LIN {X 0,Y 159.433,Z 807.885,A -85,B 0,C 180,E1 -24356.561,E2 -24356.561} C_VEL
LIN {X 0,Y 155.614,Z 816.206,A -85,B 0,C 180,E1 -24359.65,E2 -24359.65} C_VEL
LIN {X 0,Y 151.771,Z 823.644,A -85,B 0,C 180,E1 -24363.159,E2 -24363.159} C_VEL
LIN {X 0,Y 148.83,Z 828.918,A -85,B 0,C 180,E1 -24366.333,E2 -24366.333} C_VEL
LIN {X 0,Y 145.963,Z 834.064,A -85,B 0,C 180,E1 -24370.301,E2 -24370.301} C_VEL
LIN {X 0,Y 143.724,Z 838.04,A -85,B 0,C 180,E1 -24374.396,E2 -24374.396} C_VEL
LIN {X 0,Y 142.137,Z 840.967,A -85,B 0,C 180,E1 -24378.591,E2 -24378.591} C_VEL
LIN {X 0,Y 141.434,Z 842.382,A -85,B 0,C 180,E1 -24381.425,E2 -24381.425} C_VEL
LIN {X 0,Y 140.7,Z 843.984,A -85,B 0,C 180,E1 -24387.135,E2 -24387.135} C_VEL
LIN {X 0,Y 140.69,Z 844.211,A -85,B 0,C 180,E1 -24389.998,E2 -24389.998} C_VEL
LIN {X 0,Y 140.947,Z 843.425,A -85,B 0,C 180,E1 -24395.721,E2 -24395.721} C_VEL
LIN {X 0,Y 141.432,Z 842.454,A -85,B 0,C 180,E1 -24398.571,E2 -24398.571} C_VEL
LIN {X 0,Y 142.132,Z 841.08,A -85,B 0,C 180,E1 -24401.405,E2 -24401.405} C_VEL
LIN {X 0,Y 143.688,Z 838.194,A -85,B 0,C 180,E1 -24405.603,E2 -24405.603} C_VEL
LIN {X 0,Y 145.898,Z 834.266,A -85,B 0,C 180,E1 -24409.703,E2 -24409.703} C_VEL
LIN {X 0,Y 148.753,Z 829.176,A -85,B 0,C 180,E1 -24413.675,E2 -24413.675} C_VEL
LIN {X 0,Y 152.357,Z 822.754,A -85,B 0,C 180,E1 -24417.467,E2 -24417.467} C_VEL
LIN {X 0,Y 156.625,Z 814.287,A -85,B 0,C 180,E1 -24421.308,E2 -24421.308} C_VEL
LIN {X 0,Y 160.109,Z 806.58,A -85,B 0,C 180,E1 -24424.029,E2 -24424.029} C_VEL
LIN {X 0,Y 164.319,Z 796.492,A -85,B 0,C 180,E1 -24426.78,E2 -24426.78} C_VEL
LIN {X 0,Y 168.42,Z 785.143,A -85,B 0,C 180,E1 -24429.132,E2 -24429.132} C_VEL
LIN {X 0,Y 171.709,Z 773.906,A -85,B 0,C 180,E1 -24430.907,E2 -24430.907} C_VEL
LIN {X 0,Y 174.569,Z 761.518,A -85,B 0,C 180,E1 -24432.338,E2 -24432.338} C_VEL
LIN {X 0,Y 176.775,Z 748.935,A -85,B 0,C 180,E1 -24433.335,E2 -24433.335} C_VEL
LIN {X 0,Y 177.807,Z 738.757,A -85,B 0,C 180,E1 -24433.901,E2 -24433.901} C_VEL
LIN {X 0,Y 173.307,Z 740.765,A -85,B 0,C 180,E1 -24435.203,E2 -24435.203} C_VEL
LIN {X 0,Y 170.147,Z 741.611,A -85,B 0,C 180,E1 -24436.222,E2 -24436.222} C_VEL
LIN {X 0,Y 165.898,Z 744.296,A -85,B 0,C 180,E1 -24437.532,E2 -24437.532} C_VEL
LIN {X 0,Y 162.52,Z 745.361,A -85,B 0,C 180,E1 -24438.74,E2 -24438.74} C_VEL
LIN {X 0,Y 159.499,Z 745.547,A -85,B 0,C 180,E1 -24439.98,E2 -24439.98} C_VEL
LIN {X 0,Y 155.97,Z 747.642,A -85,B 0,C 180,E1 -24441.302,E2 -24441.302} C_VEL
LIN {X 0,Y 154.26,Z 748.147,A -85,B 0,C 180,E1 -24442.044,E2 -24442.044} C_VEL
LIN {X 0,Y 150.109,Z 747.859,A -85,B 0,C 180,E1 -24444.18,E2 -24444.18} C_VEL
LIN {X 0,Y 147.27,Z 749.37,A -85,B 0,C 180,E1 -24445.53,E2 -24445.53} C_VEL
LIN {X 0,Y 145.442,Z 749.393,A -85,B 0,C 180,E1 -24446.599,E2 -24446.599} C_VEL
LIN {X 0,Y 144.475,Z 748.528,A -85,B 0,C 180,E1 -24447.325,E2 -24447.325} C_VEL
LIN {X 0,Y 144.158,Z 747.052,A -85,B 0,C 180,E1 -24447.828,E2 -24447.828} C_VEL
LIN {X 0,Y 143.492,Z 754.332,A -85,B 0,C 180,E1 -24451.83,E2 -24451.83} C_VEL
LIN {X 0,Y 143.482,Z 761.799,A -85,B 0,C 180,E1 -24456.93,E2 -24456.93} C_VEL
LIN {X 0,Y 144.233,Z 767.1,A -85,B 0,C 180,E1 -24461.535,E2 -24461.535} C_VEL
LIN {X 0,Y 145.804,Z 771.093,A -85,B 0,C 180,E1 -24466.054,E2 -24466.054} C_VEL
LIN {X 0,Y 147.276,Z 773.104,A -85,B 0,C 180,E1 -24468.996,E2 -24468.996} C_VEL
LIN {X 0,Y 149.078,Z 774.683,A -85,B 0,C 180,E1 -24471.869,E2 -24471.869} C_VEL
LIN {X 0,Y 151.257,Z 775.775,A -85,B 0,C 180,E1 -24474.668,E2 -24474.668} C_VEL
LIN {X 0,Y 154.674,Z 776.543,A -85,B 0,C 180,E1 -24478.326,E2 -24478.326} C_VEL
LIN {X 0,Y 159.556,Z 776.355,A -85,B 0,C 180,E1 -24482.524,E2 -24482.524} C_VEL
LIN {X 0,Y 162.872,Z 775.642,A -85,B 0,C 180,E1 -24484.951,E2 -24484.951} C_VEL
LIN {X 0,Y 166.498,Z 774.491,A -85,B 0,C 180,E1 -24487.275,E2 -24487.275} C_VEL
LIN {X 0,Y 171.25,Z 772.464,A -85,B 0,C 180,E1 -24489.971,E2 -24489.971} C_VEL
LIN {X 0,Y 176.597,Z 769.564,A -85,B 0,C 180,E1 -24492.643,E2 -24492.643} C_VEL
LIN {X 0,Y 183.317,Z 765.026,A -85,B 0,C 180,E1 -24495.567,E2 -24495.567} C_VEL
LIN {X 0,Y 190.412,Z 759.281,A -85,B 0,C 180,E1 -24498.284,E2 -24498.284} C_VEL
LIN {X 0,Y 197.891,Z 752.001,A -85,B 0,C 180,E1 -24500.802,E2 -24500.802} C_VEL
LIN {X 0,Y 205.676,Z 742.876,A -85,B 0,C 180,E1 -24503.14,E2 -24503.14} C_VEL
LIN {X 0,Y 212.006,Z 734.049,A -85,B 0,C 180,E1 -24504.884,E2 -24504.884} C_VEL
LIN {X 0,Y 217.692,Z 724.562,A -85,B 0,C 180,E1 -24506.354,E2 -24506.354} C_VEL
LIN {X 0,Y 223.591,Z 712.612,A -85,B 0,C 180,E1 -24507.824,E2 -24507.824} C_VEL
LIN {X 0,Y 228.396,Z 700.131,A -85,B 0,C 180,E1 -24508.987,E2 -24508.987} C_VEL
LIN {X 0,Y 231.612,Z 688.931,A -85,B 0,C 180,E1 -24509.841,E2 -24509.841} C_VEL
LIN {X 0,Y 232.53,Z 684.952,A -85,B 0,C 180,E1 -24510.119,E2 -24510.119} C_VEL
LIN {X 0,Y 232.21,Z 685.318,A -85,B 0,C 180,E1 -24511.425,E2 -24511.425} C_VEL
LIN {X 0,Y 231.811,Z 686.774,A -85,B 0,C 180,E1 -24512.878,E2 -24512.878} C_VEL
LIN {X 0,Y 231.448,Z 690.251,A -85,B 0,C 180,E1 -24515.018,E2 -24515.018} C_VEL
LIN {X 0,Y 228.723,Z 701.141,A -85,B 0,C 180,E1 -24515.936,E2 -24515.936} C_VEL
LIN {X 0,Y 223.27,Z 716.625,A -85,B 0,C 180,E1 -24516.732,E2 -24516.732} C_VEL
LIN {X 0,Y 217.31,Z 729.757,A -85,B 0,C 180,E1 -24517.598,E2 -24517.598} C_VEL
LIN {X 0,Y 211.644,Z 740.071,A -85,B 0,C 180,E1 -24518.504,E2 -24518.504} C_VEL
LIN {X 0,Y 208.404,Z 744.999,A -85,B 0,C 180,E1 -24518.827,E2 -24518.827} C_VEL
LIN {X 0,Y 202.208,Z 752.79,A -85,B 0,C 180,E1 -24518.994,E2 -24518.994} C_VEL
LIN {X 0,Y 195.68,Z 759.99,A -85,B 0,C 180,E1 -24519.3,E2 -24519.3} C_VEL
LIN {X 0,Y 191.955,Z 764.049,A -85,B 0,C 180,E1 -24519.853,E2 -24519.853} C_VEL
LIN {X 0,Y 182.386,Z 774.075,A -85,B 0,C 180,E1 -24522.121,E2 -24522.121} C_VEL
LIN {X 0,Y 173.174,Z 782.415,A -85,B 0,C 180,E1 -24524.751,E2 -24524.751} C_VEL
LIN {X 0,Y 165.897,Z 788.257,A -85,B 0,C 180,E1 -24527.33,E2 -24527.33} C_VEL
LIN {X 0,Y 162.05,Z 791.386,A -85,B 0,C 180,E1 -24529.011,E2 -24529.011} C_VEL
LIN {X 0,Y 157.677,Z 802.954,A -85,B 0,C 180,E1 -24531.394,E2 -24531.394} C_VEL
LIN {X 0,Y 153.161,Z 813.235,A -85,B 0,C 180,E1 -24534.197,E2 -24534.197} C_VEL
LIN {X 0,Y 149.036,Z 821.56,A -85,B 0,C 180,E1 -24537.163,E2 -24537.163} C_VEL
LIN {X 0,Y 144.79,Z 829.691,A -85,B 0,C 180,E1 -24540.965,E2 -24540.965} C_VEL
LIN {X 0,Y 141.114,Z 836.225,A -85,B 0,C 180,E1 -24544.958,E2 -24544.958} C_VEL
LIN {X 0,Y 138.146,Z 841.42,A -85,B 0,C 180,E1 -24549.141,E2 -24549.141} C_VEL
LIN {X 0,Y 135.89,Z 845.439,A -85,B 0,C 180,E1 -24553.477,E2 -24553.477} C_VEL
LIN {X 0,Y 134.464,Z 848.406,A -85,B 0,C 180,E1 -24557.935,E2 -24557.935} C_VEL
LIN {X 0,Y 133.856,Z 849.828,A -85,B 0,C 180,E1 -24560.94,E2 -24560.94} C_VEL
LIN {X 0,Y 133.526,Z 851.454,A -85,B 0,C 180,E1 -24566.985,E2 -24566.985} C_VEL
LIN {X 0,Y 133.661,Z 851.673,A -85,B 0,C 180,E1 -24570.003,E2 -24570.003} C_VEL
LIN {X 0,Y 133.527,Z 851.438,A -85,B 0,C 180,E1 -24573.02,E2 -24573.02} C_VEL
LIN {X 0,Y 133.558,Z 850.809,A -85,B 0,C 180,E1 -24576.044,E2 -24576.044} C_VEL
LIN {X 0,Y 133.858,Z 849.789,A -85,B 0,C 180,E1 -24579.065,E2 -24579.065} C_VEL
LIN {X 0,Y 134.464,Z 848.345,A -85,B 0,C 180,E1 -24582.07,E2 -24582.07} C_VEL
LIN {X 0,Y 135.87,Z 845.356,A -85,B 0,C 180,E1 -24586.531,E2 -24586.531} C_VEL
LIN {X 0,Y 138.113,Z 841.312,A -85,B 0,C 180,E1 -24590.869,E2 -24590.869} C_VEL
LIN {X 0,Y 141.693,Z 835.082,A -85,B 0,C 180,E1 -24595.724,E2 -24595.724} C_VEL
LIN {X 0,Y 145.364,Z 828.414,A -85,B 0,C 180,E1 -24599.629,E2 -24599.629} C_VEL
LIN {X 0,Y 148.981,Z 821.355,A -85,B 0,C 180,E1 -24602.856,E2 -24602.856} C_VEL
LIN {X 0,Y 153.1,Z 812.99,A -85,B 0,C 180,E1 -24605.825,E2 -24605.825} C_VEL
LIN {X 0,Y 157.64,Z 802.637,A -85,B 0,C 180,E1 -24608.622,E2 -24608.622} C_VEL
LIN {X 0,Y 162.078,Z 790.989,A -85,B 0,C 180,E1 -24610.986,E2 -24610.986} C_VEL
LIN {X 0,Y 165.633,Z 779.257,A -85,B 0,C 180,E1 -24612.76,E2 -24612.76} C_VEL
LIN {X 0,Y 168.637,Z 767.119,A -85,B 0,C 180,E1 -24614.065,E2 -24614.065} C_VEL
LIN {X 0,Y 170.976,Z 754.448,A -85,B 0,C 180,E1 -24614.98,E2 -24614.98} C_VEL
LIN {X 0,Y 172.29,Z 740.764,A -85,B 0,C 180,E1 -24615.626,E2 -24615.626} C_VEL
LIN {X 0,Y 175.16,Z 696.8,A -85,B 0,C 180,E1 -24617.207,E2 -24617.207} C_VEL
LIN {X 0,Y 174.375,Z 675.084,A -85,B 0,C 180,E1 -24618.793,E2 -24618.793} C_VEL
LIN {X 0,Y 172.801,Z 650.948,A -85,B 0,C 180,E1 -24620.919,E2 -24620.919} C_VEL
LIN {X 0,Y 171.783,Z 647.337,A -85,B 0,C 180,E1 -24621.573,E2 -24621.573} C_VEL
LIN {X 0,Y 168.493,Z 637.862,A -85,B 0,C 180,E1 -24623.661,E2 -24623.661} C_VEL
LIN {X 0,Y 164.617,Z 631.829,A -85,B 0,C 180,E1 -24626.032,E2 -24626.032} C_VEL
LIN {X 0,Y 161.633,Z 625.28,A -85,B 0,C 180,E1 -24629.999,E2 -24629.999} C_VEL
LIN {X 0,Y 160.602,Z 623.765,A -85,B 0,C 180,E1 -24631.225,E2 -24631.225} C_VEL
LIN {X 0,Y 158.998,Z 620.197,A -85,B 0,C 180,E1 -24633.767,E2 -24633.767} C_VEL
LIN {X 0,Y 156.671,Z 616.136,A -85,B 0,C 180,E1 -24637.586,E2 -24637.586} C_VEL
LIN {X 0,Y 154.772,Z 612.752,A -85,B 0,C 180,E1 -24641.466,E2 -24641.466} C_VEL
LIN {X 0,Y 152.828,Z 609.327,A -85,B 0,C 180,E1 -24646.707,E2 -24646.707} C_VEL
LIN {X 0,Y 151.398,Z 607.318,A -85,B 0,C 180,E1 -24651.995,E2 -24651.995} C_VEL
LIN {X 0,Y 150.986,Z 606.091,A -85,B 0,C 180,E1 -24657.332,E2 -24657.332} C_VEL
LIN {X 0,Y 151.07,Z 605.988,A -85,B 0,C 180,E1 -24660,E2 -24660} C_VEL
LIN {X 0,Y 151.49,Z 607.972,A -85,B 0,C 180,E1 -24668,E2 -24668} C_VEL
LIN {X 0,Y 151.967,Z 609.157,A -85,B 0,C 180,E1 -24670.661,E2 -24670.661} C_VEL
LIN {X 0,Y 153.211,Z 612.572,A -85,B 0,C 180,E1 -24675.976,E2 -24675.976} C_VEL
LIN {X 0,Y 154.985,Z 617.053,A -85,B 0,C 180,E1 -24681.271,E2 -24681.271} C_VEL
LIN {X 0,Y 156.601,Z 621.203,A -85,B 0,C 180,E1 -24685.236,E2 -24685.236} C_VEL
LIN {X 0,Y 158.276,Z 626.514,A -85,B 0,C 180,E1 -24689.238,E2 -24689.238} C_VEL
LIN {X 0,Y 159.234,Z 629.154,A -85,B 0,C 180,E1 -24690.99,E2 -24690.99} C_VEL
LIN {X 0,Y 163.41,Z 636.139,A -85,B 0,C 180,E1 -24693.902,E2 -24693.902} C_VEL
LIN {X 0,Y 167.489,Z 643.377,A -85,B 0,C 180,E1 -24696.449,E2 -24696.449} C_VEL
LIN {X 0,Y 173.046,Z 655.01,A -85,B 0,C 180,E1 -24699.63,E2 -24699.63} C_VEL
LIN {X 0,Y 175.92,Z 662.099,A -85,B 0,C 180,E1 -24701.184,E2 -24701.184} C_VEL
LIN {X 0,Y 177.008,Z 677.278,A -85,B 0,C 180,E1 -24702.491,E2 -24702.491} C_VEL
LIN {X 0,Y 172.398,Z 741.841,A -85,B 0,C 180,E1 -24704.776,E2 -24704.776} C_VEL
LIN {X 0,Y 170.625,Z 754.436,A -85,B 0,C 180,E1 -24705.553,E2 -24705.553} C_VEL
LIN {X 0,Y 168.07,Z 767.088,A -85,B 0,C 180,E1 -24706.783,E2 -24706.783} C_VEL
LIN {X 0,Y 165.024,Z 778.4,A -85,B 0,C 180,E1 -24708.282,E2 -24708.282} C_VEL
LIN {X 0,Y 161.571,Z 788.778,A -85,B 0,C 180,E1 -24710.087,E2 -24710.087} C_VEL
LIN {X 0,Y 157.386,Z 799.406,A -85,B 0,C 180,E1 -24712.523,E2 -24712.523} C_VEL
LIN {X 0,Y 152.732,Z 809.817,A -85,B 0,C 180,E1 -24715.687,E2 -24715.687} C_VEL
LIN {X 0,Y 148.959,Z 817.482,A -85,B 0,C 180,E1 -24718.734,E2 -24718.734} C_VEL
LIN {X 0,Y 144.814,Z 824.954,A -85,B 0,C 180,E1 -24722.543,E2 -24722.543} C_VEL
LIN {X 0,Y 141.194,Z 830.953,A -85,B 0,C 180,E1 -24726.532,E2 -24726.532} C_VEL
LIN {X 0,Y 138.391,Z 835.687,A -85,B 0,C 180,E1 -24730.723,E2 -24730.723} C_VEL
LIN {X 0,Y 136.233,Z 839.302,A -85,B 0,C 180,E1 -24735.05,E2 -24735.05} C_VEL
LIN {X 0,Y 135.172,Z 841.161,A -85,B 0,C 180,E1 -24737.994,E2 -24737.994} C_VEL
LIN {X 0,Y 134.428,Z 842.575,A -85,B 0,C 180,E1 -24740.974,E2 -24740.974} C_VEL
LIN {X 0,Y 133.633,Z 844.176,A -85,B 0,C 180,E1 -24746.983,E2 -24746.983} C_VEL
LIN {X 0,Y 133.57,Z 844.347,A -85,B 0,C 180,E1 -24751.354,E2 -24751.354} C_VEL
LIN {X 0,Y 133.882,Z 843.618,A -85,B 0,C 180,E1 -24756.024,E2 -24756.024} C_VEL
LIN {X 0,Y 134.426,Z 842.646,A -85,B 0,C 180,E1 -24759.021,E2 -24759.021} C_VEL
LIN {X 0,Y 135.167,Z 841.272,A -85,B 0,C 180,E1 -24762.001,E2 -24762.001} C_VEL
LIN {X 0,Y 136.845,Z 838.386,A -85,B 0,C 180,E1 -24766.405,E2 -24766.405} C_VEL
LIN {X 0,Y 139.231,Z 834.456,A -85,B 0,C 180,E1 -24770.689,E2 -24770.689} C_VEL
LIN {X 0,Y 142.276,Z 829.365,A -85,B 0,C 180,E1 -24774.824,E2 -24774.824} C_VEL
LIN {X 0,Y 146.084,Z 822.942,A -85,B 0,C 180,E1 -24778.754,E2 -24778.754} C_VEL
LIN {X 0,Y 150.335,Z 814.98,A -85,B 0,C 180,E1 -24782.501,E2 -24782.501} C_VEL
LIN {X 0,Y 154.286,Z 806.764,A -85,B 0,C 180,E1 -24785.502,E2 -24785.502} C_VEL
LIN {X 0,Y 158.687,Z 796.672,A -85,B 0,C 180,E1 -24788.315,E2 -24788.315} C_VEL
LIN {X 0,Y 162.977,Z 785.318,A -85,B 0,C 180,E1 -24790.706,E2 -24790.706} C_VEL
LIN {X 0,Y 166.409,Z 774.073,A -85,B 0,C 180,E1 -24792.507,E2 -24792.507} C_VEL
LIN {X 0,Y 169.354,Z 761.865,A -85,B 0,C 180,E1 -24793.935,E2 -24793.935} C_VEL
LIN {X 0,Y 171.675,Z 749.194,A -85,B 0,C 180,E1 -24794.947,E2 -24794.947} C_VEL
LIN {X 0,Y 171.743,Z 747.989,A -85,B 0,C 180,E1 -24795.061,E2 -24795.061} C_VEL
LIN {X 0,Y 170.353,Z 748.631,A -85,B 0,C 180,E1 -24795.465,E2 -24795.465} C_VEL
LIN {X 0,Y 165.327,Z 751.285,A -85,B 0,C 180,E1 -24796.936,E2 -24796.936} C_VEL
LIN {X 0,Y 161.312,Z 752.281,A -85,B 0,C 180,E1 -24798.363,E2 -24798.363} C_VEL
LIN {X 0,Y 159.242,Z 752.563,A -85,B 0,C 180,E1 -24799.176,E2 -24799.176} C_VEL
LIN {X 0,Y 154.898,Z 754.619,A -85,B 0,C 180,E1 -24800.774,E2 -24800.774} C_VEL
LIN {X 0,Y 152.892,Z 755.029,A -85,B 0,C 180,E1 -24801.643,E2 -24801.643} C_VEL
LIN {X 0,Y 149.193,Z 754.991,A -85,B 0,C 180,E1 -24803.507,E2 -24803.507} C_VEL
LIN {X 0,Y 146.355,Z 756.162,A -85,B 0,C 180,E1 -24804.813,E2 -24804.813} C_VEL
LIN {X 0,Y 144.323,Z 756.378,A -85,B 0,C 180,E1 -24805.943,E2 -24805.943} C_VEL
LIN {X 0,Y 141.694,Z 755.49,A -85,B 0,C 180,E1 -24807.778,E2 -24807.778} C_VEL
LIN {X 0,Y 139.146,Z 756.562,A -85,B 0,C 180,E1 -24809.243,E2 -24809.243} C_VEL
LIN {X 0,Y 137.107,Z 756.278,A -85,B 0,C 180,E1 -24810.803,E2 -24810.803} C_VEL
LIN {X 0,Y 136.443,Z 754.919,A -85,B 0,C 180,E1 -24811.661,E2 -24811.661} C_VEL
LIN {X 0,Y 136.386,Z 754.349,A -85,B 0,C 180,E1 -24811.846,E2 -24811.846} C_VEL
LIN {X 0,Y 136.282,Z 759.966,A -85,B 0,C 180,E1 -24815.634,E2 -24815.634} C_VEL
LIN {X 0,Y 136.88,Z 765.906,A -85,B 0,C 180,E1 -24820.504,E2 -24820.504} C_VEL
LIN {X 0,Y 138.319,Z 770.505,A -85,B 0,C 180,E1 -24825.282,E2 -24825.282} C_VEL
LIN {X 0,Y 139.725,Z 772.89,A -85,B 0,C 180,E1 -24828.393,E2 -24828.393} C_VEL
LIN {X 0,Y 141.912,Z 775.165,A -85,B 0,C 180,E1 -24832.06,E2 -24832.06} C_VEL
LIN {X 0,Y 146.128,Z 777.229,A -85,B 0,C 180,E1 -24837.243,E2 -24837.243} C_VEL
LIN {X 0,Y 148.914,Z 777.777,A -85,B 0,C 180,E1 -24840,E2 -24840} C_VEL
LIN {X 0,Y 152.048,Z 777.864,A -85,B 0,C 180,E1 -24842.649,E2 -24842.649} C_VEL
LIN {X 0,Y 155.449,Z 777.501,A -85,B 0,C 180,E1 -24845.188,E2 -24845.188} C_VEL
LIN {X 0,Y 159.131,Z 776.727,A -85,B 0,C 180,E1 -24847.614,E2 -24847.614} C_VEL
LIN {X 0,Y 164.484,Z 774.951,A -85,B 0,C 180,E1 -24850.678,E2 -24850.678} C_VEL
LIN {X 0,Y 171.757,Z 771.563,A -85,B 0,C 180,E1 -24854.212,E2 -24854.212} C_VEL
LIN {X 0,Y 178.839,Z 767.322,A -85,B 0,C 180,E1 -24857.142,E2 -24857.142} C_VEL
LIN {X 0,Y 187.16,Z 761.027,A -85,B 0,C 180,E1 -24860.162,E2 -24860.162} C_VEL
LIN {X 0,Y 195.403,Z 753.555,A -85,B 0,C 180,E1 -24862.746,E2 -24862.746} C_VEL
LIN {X 0,Y 203.187,Z 744.927,A -85,B 0,C 180,E1 -24864.922,E2 -24864.922} C_VEL
LIN {X 0,Y 211.228,Z 734.197,A -85,B 0,C 180,E1 -24866.958,E2 -24866.958} C_VEL
LIN {X 0,Y 217.505,Z 723.948,A -85,B 0,C 180,E1 -24868.451,E2 -24868.451} C_VEL
LIN {X 0,Y 222.732,Z 713.501,A -85,B 0,C 180,E1 -24869.651,E2 -24869.651} C_VEL
LIN {X 0,Y 227.729,Z 700.942,A -85,B 0,C 180,E1 -24870.781,E2 -24870.781} C_VEL
LIN {X 0,Y 230.426,Z 692.352,A -85,B 0,C 180,E1 -24871.455,E2 -24871.455} C_VEL
LIN {X 0,Y 230.064,Z 693.596,A -85,B 0,C 180,E1 -24872.512,E2 -24872.512} C_VEL
LIN {X 0,Y 229.618,Z 695.562,A -85,B 0,C 180,E1 -24873.654,E2 -24873.654} C_VEL
LIN {X 0,Y 227,Z 704.287,A -85,B 0,C 180,E1 -24874.323,E2 -24874.323} C_VEL
LIN {X 0,Y 221.503,Z 718.33,A -85,B 0,C 180,E1 -24875.011,E2 -24875.011} C_VEL
LIN {X 0,Y 214.736,Z 731.889,A -85,B 0,C 180,E1 -24875.905,E2 -24875.905} C_VEL
LIN {X 0,Y 206.968,Z 744.59,A -85,B 0,C 180,E1 -24877.066,E2 -24877.066} C_VEL
LIN {X 0,Y 199.435,Z 755.069,A -85,B 0,C 180,E1 -24878.368,E2 -24878.368} C_VEL
LIN {X 0,Y 191.955,Z 764.049,A -85,B 0,C 180,E1 -24879.853,E2 -24879.853} C_VEL
LIN {X 0,Y 188.055,Z 768.042,A -85,B 0,C 180,E1 -24880.484,E2 -24880.484} C_VEL
LIN {X 0,Y 180.591,Z 774.245,A -85,B 0,C 180,E1 -24881.156,E2 -24881.156} C_VEL
LIN {X 0,Y 172.911,Z 779.836,A -85,B 0,C 180,E1 -24881.995,E2 -24881.995} C_VEL
LIN {X 0,Y 168.724,Z 782.875,A -85,B 0,C 180,E1 -24882.91,E2 -24882.91} C_VEL
LIN {X 0,Y 160.759,Z 788.694,A -85,B 0,C 180,E1 -24885.619,E2 -24885.619} C_VEL
LIN {X 0,Y 156.614,Z 791.561,A -85,B 0,C 180,E1 -24887.369,E2 -24887.369} C_VEL
LIN {X 0,Y 152.177,Z 802.773,A -85,B 0,C 180,E1 -24889.721,E2 -24889.721} C_VEL
LIN {X 0,Y 147.436,Z 813.051,A -85,B 0,C 180,E1 -24892.575,E2 -24892.575} C_VEL
LIN {X 0,Y 142.306,Z 822.849,A -85,B 0,C 180,E1 -24896.252,E2 -24896.252} C_VEL
LIN {X 0,Y 137.863,Z 830.844,A -85,B 0,C 180,E1 -24900.289,E2 -24900.289} C_VEL
LIN {X 0,Y 134.701,Z 836.035,A -85,B 0,C 180,E1 -24903.677,E2 -24903.677} C_VEL
LIN {X 0,Y 131.506,Z 841.228,A -85,B 0,C 180,E1 -24908.035,E2 -24908.035} C_VEL
LIN {X 0,Y 129.067,Z 845.246,A -85,B 0,C 180,E1 -24912.576,E2 -24912.576} C_VEL
LIN {X 0,Y 127.491,Z 848.213,A -85,B 0,C 180,E1 -24917.264,E2 -24917.264} C_VEL
LIN {X 0,Y 126.82,Z 849.635,A -85,B 0,C 180,E1 -24920.433,E2 -24920.433} C_VEL
LIN {X 0,Y 126.445,Z 851.261,A -85,B 0,C 180,E1 -24926.816,E2 -24926.816} C_VEL
LIN {X 0,Y 126.514,Z 851.446,A -85,B 0,C 180,E1 -24930.718,E2 -24930.718} C_VEL
LIN {X 0,Y 126.476,Z 850.615,A -85,B 0,C 180,E1 -24936.383,E2 -24936.383} C_VEL
LIN {X 0,Y 126.822,Z 849.595,A -85,B 0,C 180,E1 -24939.572,E2 -24939.572} C_VEL
LIN {X 0,Y 127.489,Z 848.15,A -85,B 0,C 180,E1 -24942.741,E2 -24942.741} C_VEL
LIN {X 0,Y 129.045,Z 845.162,A -85,B 0,C 180,E1 -24947.432,E2 -24947.432} C_VEL
LIN {X 0,Y 131.479,Z 841.118,A -85,B 0,C 180,E1 -24951.976,E2 -24951.976} C_VEL
LIN {X 0,Y 135.331,Z 834.889,A -85,B 0,C 180,E1 -24957.029,E2 -24957.029} C_VEL
LIN {X 0,Y 139.29,Z 828.099,A -85,B 0,C 180,E1 -24961.145,E2 -24961.145} C_VEL
LIN {X 0,Y 143.051,Z 821.164,A -85,B 0,C 180,E1 -24964.403,E2 -24964.403} C_VEL
LIN {X 0,Y 147.384,Z 812.8,A -85,B 0,C 180,E1 -24967.446,E2 -24967.446} C_VEL
LIN {X 0,Y 152.149,Z 802.45,A -85,B 0,C 180,E1 -24970.294,E2 -24970.294} C_VEL
LIN {X 0,Y 156.785,Z 790.806,A -85,B 0,C 180,E1 -24972.689,E2 -24972.689} C_VEL
LIN {X 0,Y 160.501,Z 779.079,A -85,B 0,C 180,E1 -24974.478,E2 -24974.478} C_VEL
LIN {X 0,Y 163.621,Z 766.951,A -85,B 0,C 180,E1 -24975.791,E2 -24975.791} C_VEL
LIN {X 0,Y 166.018,Z 754.47,A -85,B 0,C 180,E1 -24976.698,E2 -24976.698} C_VEL
LIN {X 0,Y 167.449,Z 740.25,A -85,B 0,C 180,E1 -24977.371,E2 -24977.371} C_VEL
LIN {X 0,Y 170.376,Z 697.159,A -85,B 0,C 180,E1 -24978.946,E2 -24978.946} C_VEL
LIN {X 0,Y 169.601,Z 673.672,A -85,B 0,C 180,E1 -24980.756,E2 -24980.756} C_VEL
LIN {X 0,Y 168.379,Z 653.086,A -85,B 0,C 180,E1 -24982.657,E2 -24982.657} C_VEL
LIN {X 0,Y 164.983,Z 642.689,A -85,B 0,C 180,E1 -24984.988,E2 -24984.988} C_VEL
LIN {X 0,Y 160.526,Z 635.959,A -85,B 0,C 180,E1 -24987.868,E2 -24987.868} C_VEL
LIN {X 0,Y 157.768,Z 631.739,A -85,B 0,C 180,E1 -24989.924,E2 -24989.924} C_VEL
LIN {X 0,Y 154.856,Z 625.663,A -85,B 0,C 180,E1 -24994.46,E2 -24994.46} C_VEL
LIN {X 0,Y 152.595,Z 621.59,A -85,B 0,C 180,E1 -24998.38,E2 -24998.38} C_VEL
LIN {X 0,Y 151.362,Z 619.266,A -85,B 0,C 180,E1 -25001.033,E2 -25001.033} C_VEL
LIN {X 0,Y 149.279,Z 615.652,A -85,B 0,C 180,E1 -25006.385,E2 -25006.385} C_VEL
LIN {X 0,Y 147.929,Z 613.563,A -85,B 0,C 180,E1 -25011.806,E2 -25011.806} C_VEL
LIN {X 0,Y 147.441,Z 612.273,A -85,B 0,C 180,E1 -25017.268,E2 -25017.268} C_VEL
LIN {X 0,Y 147.42,Z 612.095,A -85,B 0,C 180,E1 -25020,E2 -25020} C_VEL
LIN {X 0,Y 147.709,Z 614.109,A -85,B 0,C 180,E1 -25028.207,E2 -25028.207} C_VEL
LIN {X 0,Y 148.616,Z 616.961,A -85,B 0,C 180,E1 -25033.677,E2 -25033.677} C_VEL
LIN {X 0,Y 150.103,Z 621.034,A -85,B 0,C 180,E1 -25039.132,E2 -25039.132} C_VEL
LIN {X 0,Y 151.554,Z 624.94,A -85,B 0,C 180,E1 -25043.215,E2 -25043.215} C_VEL
LIN {X 0,Y 153.161,Z 629.484,A -85,B 0,C 180,E1 -25046.987,E2 -25046.987} C_VEL
LIN {X 0,Y 157.861,Z 637.183,A -85,B 0,C 180,E1 -25050.855,E2 -25050.855} C_VEL
LIN {X 0,Y 162.168,Z 644.72,A -85,B 0,C 180,E1 -25053.916,E2 -25053.916} C_VEL
LIN {X 0,Y 166.718,Z 654,A -85,B 0,C 180,E1 -25056.845,E2 -25056.845} C_VEL
LIN {X 0,Y 170.665,Z 663.158,A -85,B 0,C 180,E1 -25059.188,E2 -25059.188} C_VEL
LIN {X 0,Y 171.442,Z 665.479,A -85,B 0,C 180,E1 -25059.656,E2 -25059.656} C_VEL
LIN {X 0,Y 172.284,Z 677.342,A -85,B 0,C 180,E1 -25060.745,E2 -25060.745} C_VEL
LIN {X 0,Y 167.532,Z 741.504,A -85,B 0,C 180,E1 -25063.035,E2 -25063.035} C_VEL
LIN {X 0,Y 165.64,Z 754.6,A -85,B 0,C 180,E1 -25063.836,E2 -25063.836} C_VEL
LIN {X 0,Y 162.977,Z 767.264,A -85,B 0,C 180,E1 -25065.077,E2 -25065.077} C_VEL
LIN {X 0,Y 159.801,Z 778.581,A -85,B 0,C 180,E1 -25066.59,E2 -25066.59} C_VEL
LIN {X 0,Y 156.205,Z 788.963,A -85,B 0,C 180,E1 -25068.42,E2 -25068.42} C_VEL
LIN {X 0,Y 151.816,Z 799.594,A -85,B 0,C 180,E1 -25070.893,E2 -25070.893} C_VEL
LIN {X 0,Y 146.926,Z 810.008,A -85,B 0,C 180,E1 -25074.127,E2 -25074.127} C_VEL
LIN {X 0,Y 142.152,Z 819.012,A -85,B 0,C 180,E1 -25077.892,E2 -25077.892} C_VEL
LIN {X 0,Y 137.908,Z 826.24,A -85,B 0,C 180,E1 -25081.873,E2 -25081.873} C_VEL
LIN {X 0,Y 134.702,Z 831.146,A -85,B 0,C 180,E1 -25085.327,E2 -25085.327} C_VEL
LIN {X 0,Y 131.702,Z 835.88,A -85,B 0,C 180,E1 -25089.702,E2 -25089.702} C_VEL
LIN {X 0,Y 129.377,Z 839.495,A -85,B 0,C 180,E1 -25094.237,E2 -25094.237} C_VEL
LIN {X 0,Y 128.235,Z 841.355,A -85,B 0,C 180,E1 -25097.334,E2 -25097.334} C_VEL
LIN {X 0,Y 127.415,Z 842.768,A -85,B 0,C 180,E1 -25100.473,E2 -25100.473} C_VEL
LIN {X 0,Y 126.555,Z 844.369,A -85,B 0,C 180,E1 -25106.814,E2 -25106.814} C_VEL
LIN {X 0,Y 126.505,Z 844.597,A -85,B 0,C 180,E1 -25109.997,E2 -25109.997} C_VEL
LIN {X 0,Y 126.515,Z 844.4,A -85,B 0,C 180,E1 -25113.182,E2 -25113.182} C_VEL
LIN {X 0,Y 127.412,Z 842.839,A -85,B 0,C 180,E1 -25119.522,E2 -25119.522} C_VEL
LIN {X 0,Y 128.23,Z 841.465,A -85,B 0,C 180,E1 -25122.661,E2 -25122.661} C_VEL
LIN {X 0,Y 130.034,Z 838.578,A -85,B 0,C 180,E1 -25127.29,E2 -25127.29} C_VEL
LIN {X 0,Y 132.589,Z 834.648,A -85,B 0,C 180,E1 -25131.777,E2 -25131.777} C_VEL
LIN {X 0,Y 135.863,Z 829.555,A -85,B 0,C 180,E1 -25136.081,E2 -25136.081} C_VEL
LIN {X 0,Y 139.892,Z 823.131,A -85,B 0,C 180,E1 -25140.155,E2 -25140.155} C_VEL
LIN {X 0,Y 144.129,Z 815.654,A -85,B 0,C 180,E1 -25143.805,E2 -25143.805} C_VEL
LIN {X 0,Y 148.549,Z 806.948,A -85,B 0,C 180,E1 -25147.097,E2 -25147.097} C_VEL
LIN {X 0,Y 153.171,Z 796.852,A -85,B 0,C 180,E1 -25149.965,E2 -25149.965} C_VEL
LIN {X 0,Y 157.677,Z 785.493,A -85,B 0,C 180,E1 -25152.385,E2 -25152.385} C_VEL
LIN {X 0,Y 161.248,Z 774.239,A -85,B 0,C 180,E1 -25154.212,E2 -25154.212} C_VEL
LIN {X 0,Y 164.213,Z 762.493,A -85,B 0,C 180,E1 -25155.605,E2 -25155.605} C_VEL
LIN {X 0,Y 164.872,Z 759.472,A -85,B 0,C 180,E1 -25155.902,E2 -25155.902} C_VEL
LIN {X 0,Y 164.837,Z 758.01,A -85,B 0,C 180,E1 -25156.145,E2 -25156.145} C_VEL
LIN {X 0,Y 158.589,Z 759.444,A -85,B 0,C 180,E1 -25158.337,E2 -25158.337} C_VEL
LIN {X 0,Y 153.51,Z 761.453,A -85,B 0,C 180,E1 -25160.137,E2 -25160.137} C_VEL
LIN {X 0,Y 149.078,Z 761.696,A -85,B 0,C 180,E1 -25162.203,E2 -25162.203} C_VEL
LIN {X 0,Y 144.566,Z 762.932,A -85,B 0,C 180,E1 -25164.311,E2 -25164.311} C_VEL
LIN {X 0,Y 140.685,Z 762.736,A -85,B 0,C 180,E1 -25166.666,E2 -25166.666} C_VEL
LIN {X 0,Y 136.805,Z 763.364,A -85,B 0,C 180,E1 -25169.088,E2 -25169.088} C_VEL
LIN {X 0,Y 133.746,Z 762.181,A -85,B 0,C 180,E1 -25171.775,E2 -25171.775} C_VEL
LIN {X 0,Y 130.379,Z 762.932,A -85,B 0,C 180,E1 -25174.454,E2 -25174.454} C_VEL
LIN {X 0,Y 129.322,Z 761.702,A -85,B 0,C 180,E1 -25175.948,E2 -25175.948} C_VEL
LIN {X 0,Y 129.256,Z 760.809,A -85,B 0,C 180,E1 -25176.461,E2 -25176.461} C_VEL
LIN {X 0,Y 129.865,Z 766.248,A -85,B 0,C 180,E1 -25181.052,E2 -25181.052} C_VEL
LIN {X 0,Y 131.559,Z 771.297,A -85,B 0,C 180,E1 -25186.348,E2 -25186.348} C_VEL
LIN {X 0,Y 133.882,Z 774.659,A -85,B 0,C 180,E1 -25190.939,E2 -25190.939} C_VEL
LIN {X 0,Y 136.005,Z 776.458,A -85,B 0,C 180,E1 -25194.068,E2 -25194.068} C_VEL
LIN {X 0,Y 140.563,Z 778.488,A -85,B 0,C 180,E1 -25199.281,E2 -25199.281} C_VEL
LIN {X 0,Y 144.502,Z 779.122,A -85,B 0,C 180,E1 -25202.788,E2 -25202.788} C_VEL
LIN {X 0,Y 148.31,Z 779.089,A -85,B 0,C 180,E1 -25205.689,E2 -25205.689} C_VEL
LIN {X 0,Y 151.734,Z 778.683,A -85,B 0,C 180,E1 -25207.987,E2 -25207.987} C_VEL
LIN {X 0,Y 157.752,Z 777.23,A -85,B 0,C 180,E1 -25211.459,E2 -25211.459} C_VEL
LIN {X 0,Y 164.645,Z 774.685,A -85,B 0,C 180,E1 -25214.84,E2 -25214.84} C_VEL
LIN {X 0,Y 171.963,Z 771.028,A -85,B 0,C 180,E1 -25217.85,E2 -25217.85} C_VEL
LIN {X 0,Y 180.574,Z 765.56,A -85,B 0,C 180,E1 -25220.926,E2 -25220.926} C_VEL
LIN {X 0,Y 188.994,Z 758.942,A -85,B 0,C 180,E1 -25223.563,E2 -25223.563} C_VEL
LIN {X 0,Y 197.431,Z 750.915,A -85,B 0,C 180,E1 -25225.853,E2 -25225.853} C_VEL
LIN {X 0,Y 205.459,Z 741.705,A -85,B 0,C 180,E1 -25227.807,E2 -25227.807} C_VEL
LIN {X 0,Y 212.612,Z 731.752,A -85,B 0,C 180,E1 -25229.446,E2 -25229.446} C_VEL
LIN {X 0,Y 219.241,Z 720.541,A -85,B 0,C 180,E1 -25230.857,E2 -25230.857} C_VEL
LIN {X 0,Y 224.436,Z 709.655,A -85,B 0,C 180,E1 -25231.925,E2 -25231.925} C_VEL
LIN {X 0,Y 225.949,Z 705.881,A -85,B 0,C 180,E1 -25232.24,E2 -25232.24} C_VEL
LIN {X 0,Y 225.364,Z 707.49,A -85,B 0,C 180,E1 -25232.653,E2 -25232.653} C_VEL
LIN {X 0,Y 219.384,Z 721.166,A -85,B 0,C 180,E1 -25233.325,E2 -25233.325} C_VEL
LIN {X 0,Y 212.339,Z 734.087,A -85,B 0,C 180,E1 -25234.166,E2 -25234.166} C_VEL
LIN {X 0,Y 204.416,Z 746.084,A -85,B 0,C 180,E1 -25235.264,E2 -25235.264} C_VEL
LIN {X 0,Y 195.145,Z 757.762,A -85,B 0,C 180,E1 -25236.748,E2 -25236.748} C_VEL
LIN {X 0,Y 186.286,Z 767.447,A -85,B 0,C 180,E1 -25238.483,E2 -25238.483} C_VEL
LIN {X 0,Y 176.339,Z 776.656,A -85,B 0,C 180,E1 -25240.782,E2 -25240.782} C_VEL
LIN {X 0,Y 168.724,Z 782.875,A -85,B 0,C 180,E1 -25242.91,E2 -25242.91} C_VEL
LIN {X 0,Y 164.599,Z 785.76,A -85,B 0,C 180,E1 -25243.921,E2 -25243.921} C_VEL
LIN {X 0,Y 157.089,Z 790.755,A -85,B 0,C 180,E1 -25245.244,E2 -25245.244} C_VEL
LIN {X 0,Y 151.584,Z 795.369,A -85,B 0,C 180,E1 -25246.268,E2 -25246.268} C_VEL
LIN {X 0,Y 148.373,Z 799.439,A -85,B 0,C 180,E1 -25247.182,E2 -25247.182} C_VEL
LIN {X 0,Y 147.592,Z 800.923,A -85,B 0,C 180,E1 -25247.531,E2 -25247.531} C_VEL
LIN {X 0,Y 142.816,Z 810.957,A -85,B 0,C 180,E1 -25250.232,E2 -25250.232} C_VEL
LIN {X 0,Y 138.153,Z 819.646,A -85,B 0,C 180,E1 -25253.296,E2 -25253.296} C_VEL
LIN {X 0,Y 134.025,Z 826.814,A -85,B 0,C 180,E1 -25256.595,E2 -25256.595} C_VEL
LIN {X 0,Y 129.75,Z 833.841,A -85,B 0,C 180,E1 -25260.828,E2 -25260.828} C_VEL
LIN {X 0,Y 125.999,Z 839.43,A -85,B 0,C 180,E1 -25265.274,E2 -25265.274} C_VEL
LIN {X 0,Y 123.022,Z 843.815,A -85,B 0,C 180,E1 -25269.958,E2 -25269.958} C_VEL
LIN {X 0,Y 121.624,Z 846.132,A -85,B 0,C 180,E1 -25273.21,E2 -25273.21} C_VEL
LIN {X 0,Y 120.547,Z 848.02,A -85,B 0,C 180,E1 -25276.517,E2 -25276.517} C_VEL
LIN {X 0,Y 119.808,Z 849.442,A -85,B 0,C 180,E1 -25279.867,E2 -25279.867} C_VEL
LIN {X 0,Y 119.356,Z 851.068,A -85,B 0,C 180,E1 -25286.627,E2 -25286.627} C_VEL
LIN {X 0,Y 119.476,Z 851.287,A -85,B 0,C 180,E1 -25290.003,E2 -25290.003} C_VEL
LIN {X 0,Y 119.357,Z 851.052,A -85,B 0,C 180,E1 -25293.378,E2 -25293.378} C_VEL
LIN {X 0,Y 119.81,Z 849.401,A -85,B 0,C 180,E1 -25300.138,E2 -25300.138} C_VEL
LIN {X 0,Y 120.545,Z 847.956,A -85,B 0,C 180,E1 -25303.489,E2 -25303.489} C_VEL
LIN {X 0,Y 122.239,Z 844.967,A -85,B 0,C 180,E1 -25308.437,E2 -25308.437} C_VEL
LIN {X 0,Y 124.903,Z 840.924,A -85,B 0,C 180,E1 -25313.198,E2 -25313.198} C_VEL
LIN {X 0,Y 129.046,Z 834.697,A -85,B 0,C 180,E1 -25318.462,E2 -25318.462} C_VEL
LIN {X 0,Y 133.229,Z 827.906,A -85,B 0,C 180,E1 -25322.734,E2 -25322.734} C_VEL
LIN {X 0,Y 137.221,Z 820.972,A -85,B 0,C 180,E1 -25326.088,E2 -25326.088} C_VEL
LIN {X 0,Y 141.8,Z 812.61,A -85,B 0,C 180,E1 -25329.195,E2 -25329.195} C_VEL
LIN {X 0,Y 146.797,Z 802.263,A -85,B 0,C 180,E1 -25332.089,E2 -25332.089} C_VEL
LIN {X 0,Y 151.646,Z 790.622,A -85,B 0,C 180,E1 -25334.507,E2 -25334.507} C_VEL
LIN {X 0,Y 155.518,Z 778.902,A -85,B 0,C 180,E1 -25336.309,E2 -25336.309} C_VEL
LIN {X 0,Y 158.762,Z 766.782,A -85,B 0,C 180,E1 -25337.624,E2 -25337.624} C_VEL
LIN {X 0,Y 161.21,Z 754.475,A -85,B 0,C 180,E1 -25338.524,E2 -25338.524} C_VEL
LIN {X 0,Y 162.668,Z 740.918,A -85,B 0,C 180,E1 -25339.181,E2 -25339.181} C_VEL
LIN {X 0,Y 165.757,Z 698.112,A -85,B 0,C 180,E1 -25340.744,E2 -25340.744} C_VEL
LIN {X 0,Y 165.144,Z 674.866,A -85,B 0,C 180,E1 -25342.6,E2 -25342.6} C_VEL
LIN {X 0,Y 164.181,Z 656.067,A -85,B 0,C 180,E1 -25344.395,E2 -25344.395} C_VEL
LIN {X 0,Y 161.509,Z 647.555,A -85,B 0,C 180,E1 -25346.398,E2 -25346.398} C_VEL
LIN {X 0,Y 157.373,Z 641.115,A -85,B 0,C 180,E1 -25349.284,E2 -25349.284} C_VEL
LIN {X 0,Y 154.006,Z 636.151,A -85,B 0,C 180,E1 -25351.93,E2 -25351.93} C_VEL
LIN {X 0,Y 150.858,Z 631.46,A -85,B 0,C 180,E1 -25354.843,E2 -25354.843} C_VEL
LIN {X 0,Y 148.516,Z 627.06,A -85,B 0,C 180,E1 -25359.212,E2 -25359.212} C_VEL
LIN {X 0,Y 146.789,Z 623.833,A -85,B 0,C 180,E1 -25363.306,E2 -25363.306} C_VEL
LIN {X 0,Y 145.831,Z 622.092,A -85,B 0,C 180,E1 -25366.057,E2 -25366.057} C_VEL
LIN {X 0,Y 144.323,Z 619.736,A -85,B 0,C 180,E1 -25371.6,E2 -25371.6} C_VEL
LIN {X 0,Y 143.786,Z 618.369,A -85,B 0,C 180,E1 -25377.199,E2 -25377.199} C_VEL
LIN {X 0,Y 143.757,Z 618.198,A -85,B 0,C 180,E1 -25380,E2 -25380} C_VEL
LIN {X 0,Y 143.955,Z 620.292,A -85,B 0,C 180,E1 -25388.422,E2 -25388.422} C_VEL
LIN {X 0,Y 144.836,Z 623.303,A -85,B 0,C 180,E1 -25394.041,E2 -25394.041} C_VEL
LIN {X 0,Y 146.255,Z 627.546,A -85,B 0,C 180,E1 -25399.656,E2 -25399.656} C_VEL
LIN {X 0,Y 147.075,Z 629.686,A -85,B 0,C 180,E1 -25401.878,E2 -25401.878} C_VEL
LIN {X 0,Y 151.223,Z 636.189,A -85,B 0,C 180,E1 -25406.22,E2 -25406.22} C_VEL
LIN {X 0,Y 155.282,Z 643.108,A -85,B 0,C 180,E1 -25409.765,E2 -25409.765} C_VEL
LIN {X 0,Y 159.235,Z 650.403,A -85,B 0,C 180,E1 -25412.776,E2 -25412.776} C_VEL
LIN {X 0,Y 163.967,Z 660.525,A -85,B 0,C 180,E1 -25416.018,E2 -25416.018} C_VEL
LIN {X 0,Y 167.032,Z 668.236,A -85,B 0,C 180,E1 -25417.978,E2 -25417.978} C_VEL
LIN {X 0,Y 167.67,Z 678.597,A -85,B 0,C 180,E1 -25418.957,E2 -25418.957} C_VEL
LIN {X 0,Y 162.673,Z 742.465,A -85,B 0,C 180,E1 -25421.241,E2 -25421.241} C_VEL
LIN {X 0,Y 160.655,Z 755.485,A -85,B 0,C 180,E1 -25422.069,E2 -25422.069} C_VEL
LIN {X 0,Y 157.739,Z 768.523,A -85,B 0,C 180,E1 -25423.379,E2 -25423.379} C_VEL
LIN {X 0,Y 154.171,Z 780.416,A -85,B 0,C 180,E1 -25425.041,E2 -25425.041} C_VEL
LIN {X 0,Y 149.938,Z 791.692,A -85,B 0,C 180,E1 -25427.181,E2 -25427.181} C_VEL
LIN {X 0,Y 145.426,Z 801.869,A -85,B 0,C 180,E1 -25429.729,E2 -25429.729} C_VEL
LIN {X 0,Y 141.239,Z 810.198,A -85,B 0,C 180,E1 -25432.44,E2 -25432.44} C_VEL
LIN {X 0,Y 136.176,Z 819.204,A -85,B 0,C 180,E1 -25436.3,E2 -25436.3} C_VEL
LIN {X 0,Y 131.677,Z 826.433,A -85,B 0,C 180,E1 -25440.414,E2 -25440.414} C_VEL
LIN {X 0,Y 127.141,Z 833.063,A -85,B 0,C 180,E1 -25445.505,E2 -25445.505} C_VEL
LIN {X 0,Y 124.13,Z 837.406,A -85,B 0,C 180,E1 -25450.138,E2 -25450.138} C_VEL
LIN {X 0,Y 122.557,Z 839.689,A -85,B 0,C 180,E1 -25453.335,E2 -25453.335} C_VEL
LIN {X 0,Y 121.328,Z 841.548,A -85,B 0,C 180,E1 -25456.6,E2 -25456.6} C_VEL
LIN {X 0,Y 120.43,Z 842.961,A -85,B 0,C 180,E1 -25459.914,E2 -25459.914} C_VEL
LIN {X 0,Y 119.484,Z 844.562,A -85,B 0,C 180,E1 -25466.625,E2 -25466.625} C_VEL
LIN {X 0,Y 119.419,Z 844.79,A -85,B 0,C 180,E1 -25469.997,E2 -25469.997} C_VEL
LIN {X 0,Y 119.439,Z 844.593,A -85,B 0,C 180,E1 -25473.37,E2 -25473.37} C_VEL
LIN {X 0,Y 120.427,Z 843.031,A -85,B 0,C 180,E1 -25480.08,E2 -25480.08} C_VEL
LIN {X 0,Y 121.322,Z 841.656,A -85,B 0,C 180,E1 -25483.395,E2 -25483.395} C_VEL
LIN {X 0,Y 123.259,Z 838.769,A -85,B 0,C 180,E1 -25488.273,E2 -25488.273} C_VEL
LIN {X 0,Y 125.999,Z 834.839,A -85,B 0,C 180,E1 -25492.979,E2 -25492.979} C_VEL
LIN {X 0,Y 129.526,Z 829.744,A -85,B 0,C 180,E1 -25497.462,E2 -25497.462} C_VEL
LIN {X 0,Y 133.792,Z 823.319,A -85,B 0,C 180,E1 -25501.684,E2 -25501.684} C_VEL
LIN {X 0,Y 138.002,Z 816.33,A -85,B 0,C 180,E1 -25505.225,E2 -25505.225} C_VEL
LIN {X 0,Y 142.955,Z 807.132,A -85,B 0,C 180,E1 -25508.812,E2 -25508.812} C_VEL
LIN {X 0,Y 147.809,Z 797.032,A -85,B 0,C 180,E1 -25511.73,E2 -25511.73} C_VEL
LIN {X 0,Y 152.512,Z 785.668,A -85,B 0,C 180,E1 -25514.182,E2 -25514.182} C_VEL
LIN {X 0,Y 156.256,Z 774.404,A -85,B 0,C 180,E1 -25516.021,E2 -25516.021} C_VEL
LIN {X 0,Y 158.198,Z 767.491,A -85,B 0,C 180,E1 -25516.884,E2 -25516.884} C_VEL
LIN {X 0,Y 158.025,Z 765.922,A -85,B 0,C 180,E1 -25517.294,E2 -25517.294} C_VEL
LIN {X 0,Y 151.6,Z 768.081,A -85,B 0,C 180,E1 -25519.531,E2 -25519.531} C_VEL
LIN {X 0,Y 147.074,Z 768.435,A -85,B 0,C 180,E1 -25521.595,E2 -25521.595} C_VEL
LIN {X 0,Y 142.506,Z 769.538,A -85,B 0,C 180,E1 -25523.714,E2 -25523.714} C_VEL
LIN {X 0,Y 138.572,Z 769.373,A -85,B 0,C 180,E1 -25526.09,E2 -25526.09} C_VEL
LIN {X 0,Y 134.623,Z 769.981,A -85,B 0,C 180,E1 -25528.53,E2 -25528.53} C_VEL
LIN {X 0,Y 131.525,Z 768.913,A -85,B 0,C 180,E1 -25531.255,E2 -25531.255} C_VEL
LIN {X 0,Y 128.114,Z 769.566,A -85,B 0,C 180,E1 -25533.969,E2 -25533.969} C_VEL
LIN {X 0,Y 125.701,Z 768.349,A -85,B 0,C 180,E1 -25536.96,E2 -25536.96} C_VEL
LIN {X 0,Y 123.24,Z 768.192,A -85,B 0,C 180,E1 -25539.991,E2 -25539.991} C_VEL
LIN {X 0,Y 122.832,Z 767.022,A -85,B 0,C 180,E1 -25541.225,E2 -25541.225} C_VEL
LIN {X 0,Y 122.84,Z 766.437,A -85,B 0,C 180,E1 -25541.551,E2 -25541.551} C_VEL
LIN {X 0,Y 124.611,Z 771.535,A -85,B 0,C 180,E1 -25546.962,E2 -25546.962} C_VEL
LIN {X 0,Y 127.56,Z 775.685,A -85,B 0,C 180,E1 -25552.596,E2 -25552.596} C_VEL
LIN {X 0,Y 130.827,Z 778.055,A -85,B 0,C 180,E1 -25556.92,E2 -25556.92} C_VEL
LIN {X 0,Y 133.655,Z 779.306,A -85,B 0,C 180,E1 -25560,E2 -25560} C_VEL
LIN {X 0,Y 136.89,Z 780.107,A -85,B 0,C 180,E1 -25562.943,E2 -25562.943} C_VEL
LIN {X 0,Y 141.455,Z 780.473,A -85,B 0,C 180,E1 -25566.479,E2 -25566.479} C_VEL
LIN {X 0,Y 148.456,Z 779.869,A -85,B 0,C 180,E1 -25570.915,E2 -25570.915} C_VEL
LIN {X 0,Y 152.871,Z 778.894,A -85,B 0,C 180,E1 -25573.289,E2 -25573.289} C_VEL
LIN {X 0,Y 157.555,Z 777.478,A -85,B 0,C 180,E1 -25575.524,E2 -25575.524} C_VEL
LIN {X 0,Y 165.053,Z 774.446,A -85,B 0,C 180,E1 -25578.624,E2 -25578.624} C_VEL
LIN {X 0,Y 174.132,Z 769.628,A -85,B 0,C 180,E1 -25581.839,E2 -25581.839} C_VEL
LIN {X 0,Y 182.574,Z 763.912,A -85,B 0,C 180,E1 -25584.444,E2 -25584.444} C_VEL
LIN {X 0,Y 191.268,Z 756.86,A -85,B 0,C 180,E1 -25586.751,E2 -25586.751} C_VEL
LIN {X 0,Y 198.691,Z 749.608,A -85,B 0,C 180,E1 -25588.524,E2 -25588.524} C_VEL
LIN {X 0,Y 206.959,Z 739.951,A -85,B 0,C 180,E1 -25590.329,E2 -25590.329} C_VEL
LIN {X 0,Y 213.857,Z 730.26,A -85,B 0,C 180,E1 -25591.723,E2 -25591.723} C_VEL
LIN {X 0,Y 212.904,Z 731.903,A -85,B 0,C 180,E1 -25592.083,E2 -25592.083} C_VEL
LIN {X 0,Y 204.465,Z 744.357,A -85,B 0,C 180,E1 -25593.093,E2 -25593.093} C_VEL
LIN {X 0,Y 195.751,Z 755.198,A -85,B 0,C 180,E1 -25594.338,E2 -25594.338} C_VEL
LIN {X 0,Y 186.486,Z 765.002,A -85,B 0,C 180,E1 -25595.883,E2 -25595.883} C_VEL
LIN {X 0,Y 176.133,Z 774.381,A -85,B 0,C 180,E1 -25598,E2 -25598} C_VEL
LIN {X 0,Y 166.26,Z 782.042,A -85,B 0,C 180,E1 -25600.462,E2 -25600.462} C_VEL
LIN {X 0,Y 155.776,Z 789.052,A -85,B 0,C 180,E1 -25603.796,E2 -25603.796} C_VEL
LIN {X 0,Y 151.331,Z 791.763,A -85,B 0,C 180,E1 -25605.616,E2 -25605.616} C_VEL
LIN {X 0,Y 147.592,Z 800.923,A -85,B 0,C 180,E1 -25607.531,E2 -25607.531} C_VEL
LIN {X 0,Y 144.919,Z 805.64,A -85,B 0,C 180,E1 -25608.531,E2 -25608.531} C_VEL
LIN {X 0,Y 139.032,Z 812.886,A -85,B 0,C 180,E1 -25609.935,E2 -25609.935} C_VEL
LIN {X 0,Y 133.007,Z 819.538,A -85,B 0,C 180,E1 -25611.661,E2 -25611.661} C_VEL
LIN {X 0,Y 130.183,Z 823.312,A -85,B 0,C 180,E1 -25613.164,E2 -25613.164} C_VEL
LIN {X 0,Y 125,Z 831.464,A -85,B 0,C 180,E1 -25617.721,E2 -25617.721} C_VEL
LIN {X 0,Y 120.749,Z 837.504,A -85,B 0,C 180,E1 -25622.253,E2 -25622.253} C_VEL
LIN {X 0,Y 117.355,Z 842.284,A -85,B 0,C 180,E1 -25627.095,E2 -25627.095} C_VEL
LIN {X 0,Y 114.792,Z 845.939,A -85,B 0,C 180,E1 -25632.178,E2 -25632.178} C_VEL
LIN {X 0,Y 113.635,Z 847.827,A -85,B 0,C 180,E1 -25635.68,E2 -25635.68} C_VEL
LIN {X 0,Y 112.797,Z 849.248,A -85,B 0,C 180,E1 -25639.23,E2 -25639.23} C_VEL
LIN {X 0,Y 112.263,Z 850.875,A -85,B 0,C 180,E1 -25646.414,E2 -25646.414} C_VEL
LIN {X 0,Y 112.372,Z 851.094,A -85,B 0,C 180,E1 -25650.003,E2 -25650.003} C_VEL
LIN {X 0,Y 112.264,Z 850.858,A -85,B 0,C 180,E1 -25653.592,E2 -25653.592} C_VEL
LIN {X 0,Y 112.798,Z 849.207,A -85,B 0,C 180,E1 -25660.776,E2 -25660.776} C_VEL
LIN {X 0,Y 113.632,Z 847.762,A -85,B 0,C 180,E1 -25664.326,E2 -25664.326} C_VEL
LIN {X 0,Y 115.488,Z 844.773,A -85,B 0,C 180,E1 -25669.557,E2 -25669.557} C_VEL
LIN {X 0,Y 118.393,Z 840.731,A -85,B 0,C 180,E1 -25674.555,E2 -25674.555} C_VEL
LIN {X 0,Y 122.845,Z 834.504,A -85,B 0,C 180,E1 -25680.042,E2 -25680.042} C_VEL
LIN {X 0,Y 127.274,Z 827.713,A -85,B 0,C 180,E1 -25684.474,E2 -25684.474} C_VEL
LIN {X 0,Y 131.541,Z 820.781,A -85,B 0,C 180,E1 -25687.913,E2 -25687.913} C_VEL
LIN {X 0,Y 136.365,Z 812.421,A -85,B 0,C 180,E1 -25691.082,E2 -25691.082} C_VEL
LIN {X 0,Y 141.599,Z 802.075,A -85,B 0,C 180,E1 -25694.019,E2 -25694.019} C_VEL
LIN {X 0,Y 146.084,Z 791.846,A -85,B 0,C 180,E1 -25696.193,E2 -25696.193} C_VEL
LIN {X 0,Y 150.124,Z 780.64,A -85,B 0,C 180,E1 -25698.006,E2 -25698.006} C_VEL
LIN {X 0,Y 153.464,Z 769.13,A -85,B 0,C 180,E1 -25699.334,E2 -25699.334} C_VEL
LIN {X 0,Y 156.271,Z 756.169,A -85,B 0,C 180,E1 -25700.352,E2 -25700.352} C_VEL
LIN {X 0,Y 157.869,Z 743.75,A -85,B 0,C 180,E1 -25701.018,E2 -25701.018} C_VEL
LIN {X 0,Y 161.288,Z 698.705,A -85,B 0,C 180,E1 -25702.68,E2 -25702.68} C_VEL
LIN {X 0,Y 160.829,Z 674.625,A -85,B 0,C 180,E1 -25704.67,E2 -25704.67} C_VEL
LIN {X 0,Y 160.11,Z 658.895,A -85,B 0,C 180,E1 -25706.253,E2 -25706.253} C_VEL
LIN {X 0,Y 158.243,Z 652.579,A -85,B 0,C 180,E1 -25707.795,E2 -25707.795} C_VEL
LIN {X 0,Y 153.795,Z 645.372,A -85,B 0,C 180,E1 -25711.193,E2 -25711.193} C_VEL
LIN {X 0,Y 151.449,Z 641.966,A -85,B 0,C 180,E1 -25713.192,E2 -25713.192} C_VEL
LIN {X 0,Y 148.071,Z 636.885,A -85,B 0,C 180,E1 -25716.491,E2 -25716.491} C_VEL
LIN {X 0,Y 143.701,Z 631.102,A -85,B 0,C 180,E1 -25721.833,E2 -25721.833} C_VEL
LIN {X 0,Y 142.345,Z 628.53,A -85,B 0,C 180,E1 -25725.708,E2 -25725.708} C_VEL
LIN {X 0,Y 141.535,Z 627.093,A -85,B 0,C 180,E1 -25728.544,E2 -25728.544} C_VEL
LIN {X 0,Y 140.4,Z 625.24,A -85,B 0,C 180,E1 -25734.254,E2 -25734.254} C_VEL
LIN {X 0,Y 140.237,Z 624.533,A -85,B 0,C 180,E1 -25737.128,E2 -25737.128} C_VEL
LIN {X 0,Y 140.108,Z 624.319,A -85,B 0,C 180,E1 -25740,E2 -25740} C_VEL
LIN {X 0,Y 140.11,Z 626.289,A -85,B 0,C 180,E1 -25747.968,E2 -25747.968} C_VEL
LIN {X 0,Y 140.56,Z 627.892,A -85,B 0,C 180,E1 -25751.537,E2 -25751.537} C_VEL
LIN {X 0,Y 141.34,Z 630.269,A -85,B 0,C 180,E1 -25755.133,E2 -25755.133} C_VEL
LIN {X 0,Y 145.448,Z 636.387,A -85,B 0,C 180,E1 -25761.137,E2 -25761.137} C_VEL
LIN {X 0,Y 148.933,Z 642.148,A -85,B 0,C 180,E1 -25765.039,E2 -25765.039} C_VEL
LIN {X 0,Y 152.731,Z 648.965,A -85,B 0,C 180,E1 -25768.611,E2 -25768.611} C_VEL
LIN {X 0,Y 156.857,Z 657.104,A -85,B 0,C 180,E1 -25771.97,E2 -25771.97} C_VEL
LIN {X 0,Y 160.761,Z 666.01,A -85,B 0,C 180,E1 -25774.834,E2 -25774.834} C_VEL
LIN {X 0,Y 162.845,Z 671.823,A -85,B 0,C 180,E1 -25776.306,E2 -25776.306} C_VEL
LIN {X 0,Y 163.228,Z 679.867,A -85,B 0,C 180,E1 -25777.07,E2 -25777.07} C_VEL
LIN {X 0,Y 158.117,Z 742.351,A -85,B 0,C 180,E1 -25779.298,E2 -25779.298} C_VEL
LIN {X 0,Y 156.172,Z 754.927,A -85,B 0,C 180,E1 -25780.088,E2 -25780.088} C_VEL
LIN {X 0,Y 153.28,Z 767.613,A -85,B 0,C 180,E1 -25781.337,E2 -25781.337} C_VEL
LIN {X 0,Y 149.812,Z 778.943,A -85,B 0,C 180,E1 -25782.859,E2 -25782.859} C_VEL
LIN {X 0,Y 145.92,Z 789.332,A -85,B 0,C 180,E1 -25784.729,E2 -25784.729} C_VEL
LIN {X 0,Y 141.078,Z 799.97,A -85,B 0,C 180,E1 -25787.252,E2 -25787.252} C_VEL
LIN {X 0,Y 136.614,Z 808.646,A -85,B 0,C 180,E1 -25789.978,E2 -25789.978} C_VEL
LIN {X 0,Y 132.354,Z 816.128,A -85,B 0,C 180,E1 -25793.002,E2 -25793.002} C_VEL
LIN {X 0,Y 127.099,Z 824.412,A -85,B 0,C 180,E1 -25797.373,E2 -25797.373} C_VEL
LIN {X 0,Y 123.339,Z 829.689,A -85,B 0,C 180,E1 -25801.028,E2 -25801.028} C_VEL
LIN {X 0,Y 119.54,Z 834.839,A -85,B 0,C 180,E1 -25805.696,E2 -25805.696} C_VEL
LIN {X 0,Y 116.56,Z 838.815,A -85,B 0,C 180,E1 -25810.63,E2 -25810.63} C_VEL
LIN {X 0,Y 114.424,Z 841.741,A -85,B 0,C 180,E1 -25815.775,E2 -25815.775} C_VEL
LIN {X 0,Y 113.432,Z 843.155,A -85,B 0,C 180,E1 -25819.285,E2 -25819.285} C_VEL
LIN {X 0,Y 112.416,Z 844.755,A -85,B 0,C 180,E1 -25826.413,E2 -25826.413} C_VEL
LIN {X 0,Y 112.335,Z 844.982,A -85,B 0,C 180,E1 -25829.997,E2 -25829.997} C_VEL
LIN {X 0,Y 112.746,Z 844.195,A -85,B 0,C 180,E1 -25837.159,E2 -25837.159} C_VEL
LIN {X 0,Y 113.429,Z 843.224,A -85,B 0,C 180,E1 -25840.709,E2 -25840.709} C_VEL
LIN {X 0,Y 114.418,Z 841.849,A -85,B 0,C 180,E1 -25844.22,E2 -25844.22} C_VEL
LIN {X 0,Y 116.532,Z 838.961,A -85,B 0,C 180,E1 -25849.369,E2 -25849.369} C_VEL
LIN {X 0,Y 119.473,Z 835.03,A -85,B 0,C 180,E1 -25854.313,E2 -25854.313} C_VEL
LIN {X 0,Y 123.273,Z 829.934,A -85,B 0,C 180,E1 -25858.983,E2 -25858.983} C_VEL
LIN {X 0,Y 127.797,Z 823.507,A -85,B 0,C 180,E1 -25863.359,E2 -25863.359} C_VEL
LIN {X 0,Y 132.991,Z 815.294,A -85,B 0,C 180,E1 -25867.562,E2 -25867.562} C_VEL
LIN {X 0,Y 137.497,Z 807.316,A -85,B 0,C 180,E1 -25870.666,E2 -25870.666} C_VEL
LIN {X 0,Y 142.59,Z 797.212,A -85,B 0,C 180,E1 -25873.629,E2 -25873.629} C_VEL
LIN {X 0,Y 147.406,Z 786.105,A -85,B 0,C 180,E1 -25876.05,E2 -25876.05} C_VEL
LIN {X 0,Y 151.429,Z 774.57,A -85,B 0,C 180,E1 -25877.947,E2 -25877.947} C_VEL
LIN {X 0,Y 144.812,Z 775,A -85,B 0,C 180,E1 -25880.882,E2 -25880.882} C_VEL
LIN {X 0,Y 140.167,Z 775.985,A -85,B 0,C 180,E1 -25883.009,E2 -25883.009} C_VEL
LIN {X 0,Y 136.176,Z 775.854,A -85,B 0,C 180,E1 -25885.409,E2 -25885.409} C_VEL
LIN {X 0,Y 132.138,Z 776.435,A -85,B 0,C 180,E1 -25887.868,E2 -25887.868} C_VEL
LIN {X 0,Y 129,Z 775.492,A -85,B 0,C 180,E1 -25890.638,E2 -25890.638} C_VEL
LIN {X 0,Y 125.548,Z 776.034,A -85,B 0,C 180,E1 -25893.395,E2 -25893.395} C_VEL
LIN {X 0,Y 123.08,Z 774.962,A -85,B 0,C 180,E1 -25896.44,E2 -25896.44} C_VEL
LIN {X 0,Y 120.623,Z 774.708,A -85,B 0,C 180,E1 -25899.538,E2 -25899.538} C_VEL
LIN {X 0,Y 117.454,Z 772.78,A -85,B 0,C 180,E1 -25906.152,E2 -25906.152} C_VEL
LIN {X 0,Y 117.547,Z 771.492,A -85,B 0,C 180,E1 -25907.373,E2 -25907.373} C_VEL
LIN {X 0,Y 120.652,Z 775.982,A -85,B 0,C 180,E1 -25913.31,E2 -25913.31} C_VEL
LIN {X 0,Y 123.128,Z 778.025,A -85,B 0,C 180,E1 -25916.728,E2 -25916.728} C_VEL
LIN {X 0,Y 126.501,Z 779.866,A -85,B 0,C 180,E1 -25920.513,E2 -25920.513} C_VEL
LIN {X 0,Y 132.869,Z 781.493,A -85,B 0,C 180,E1 -25926.072,E2 -25926.072} C_VEL
LIN {X 0,Y 136.798,Z 781.776,A -85,B 0,C 180,E1 -25928.866,E2 -25928.866} C_VEL
LIN {X 0,Y 144.47,Z 781.237,A -85,B 0,C 180,E1 -25933.374,E2 -25933.374} C_VEL
LIN {X 0,Y 150.412,Z 779.991,A -85,B 0,C 180,E1 -25936.281,E2 -25936.281} C_VEL
LIN {X 0,Y 155.62,Z 778.487,A -85,B 0,C 180,E1 -25938.499,E2 -25938.499} C_VEL
LIN {X 0,Y 163.464,Z 775.404,A -85,B 0,C 180,E1 -25941.435,E2 -25941.435} C_VEL
LIN {X 0,Y 171.877,Z 771.112,A -85,B 0,C 180,E1 -25944.136,E2 -25944.136} C_VEL
LIN {X 0,Y 180.878,Z 765.405,A -85,B 0,C 180,E1 -25946.669,E2 -25946.669} C_VEL
LIN {X 0,Y 189.605,Z 758.606,A -85,B 0,C 180,E1 -25948.807,E2 -25948.807} C_VEL
LIN {X 0,Y 198.446,Z 750.414,A -85,B 0,C 180,E1 -25950.714,E2 -25950.714} C_VEL
LIN {X 0,Y 200.876,Z 747.831,A -85,B 0,C 180,E1 -25951.202,E2 -25951.202} C_VEL
LIN {X 0,Y 199.548,Z 749.485,A -85,B 0,C 180,E1 -25951.576,E2 -25951.576} C_VEL
LIN {X 0,Y 190.261,Z 759.591,A -85,B 0,C 180,E1 -25952.827,E2 -25952.827} C_VEL
LIN {X 0,Y 180.934,Z 768.398,A -85,B 0,C 180,E1 -25954.374,E2 -25954.374} C_VEL
LIN {X 0,Y 170.405,Z 776.816,A -85,B 0,C 180,E1 -25956.468,E2 -25956.468} C_VEL
LIN {X 0,Y 158.98,Z 784.629,A -85,B 0,C 180,E1 -25959.325,E2 -25959.325} C_VEL
LIN {X 0,Y 150.963,Z 789.3,A -85,B 0,C 180,E1 -25961.856,E2 -25961.856} C_VEL
LIN {X 0,Y 146.199,Z 791.911,A -85,B 0,C 180,E1 -25963.737,E2 -25963.737} C_VEL
LIN {X 0,Y 141.621,Z 802.412,A -85,B 0,C 180,E1 -25965.997,E2 -25965.997} C_VEL
LIN {X 0,Y 136.407,Z 812.682,A -85,B 0,C 180,E1 -25968.939,E2 -25968.939} C_VEL
LIN {X 0,Y 130.692,Z 822.474,A -85,B 0,C 180,E1 -25972.777,E2 -25972.777} C_VEL
LIN {X 0,Y 130.183,Z 823.312,A -85,B 0,C 180,E1 -25973.164,E2 -25973.164} C_VEL
LIN {X 0,Y 127.365,Z 826.95,A -85,B 0,C 180,E1 -25974.821,E2 -25974.821} C_VEL
LIN {X 0,Y 121.273,Z 832.357,A -85,B 0,C 180,E1 -25977.445,E2 -25977.445} C_VEL
LIN {X 0,Y 115.285,Z 837.094,A -85,B 0,C 180,E1 -25980.531,E2 -25980.531} C_VEL
LIN {X 0,Y 112.727,Z 839.653,A -85,B 0,C 180,E1 -25982.884,E2 -25982.884} C_VEL
LIN {X 0,Y 108.819,Z 844.669,A -85,B 0,C 180,E1 -25989.197,E2 -25989.197} C_VEL
LIN {X 0,Y 106.739,Z 847.634,A -85,B 0,C 180,E1 -25994.733,E2 -25994.733} C_VEL
LIN {X 0,Y 105.814,Z 849.055,A -85,B 0,C 180,E1 -25998.51,E2 -25998.51} C_VEL
LIN {X 0,Y 105.156,Z 850.682,A -85,B 0,C 180,E1 -26006.171,E2 -26006.171} C_VEL
LIN {X 0,Y 105.277,Z 850.901,A -85,B 0,C 180,E1 -26010.003,E2 -26010.003} C_VEL
LIN {X 0,Y 105.157,Z 850.664,A -85,B 0,C 180,E1 -26013.835,E2 -26013.835} C_VEL
LIN {X 0,Y 105.816,Z 849.013,A -85,B 0,C 180,E1 -26021.496,E2 -26021.496} C_VEL
LIN {X 0,Y 106.736,Z 847.568,A -85,B 0,C 180,E1 -26025.274,E2 -26025.274} C_VEL
LIN {X 0,Y 108.797,Z 844.578,A -85,B 0,C 180,E1 -26030.814,E2 -26030.814} C_VEL
LIN {X 0,Y 111.956,Z 840.537,A -85,B 0,C 180,E1 -26036.07,E2 -26036.07} C_VEL
LIN {X 0,Y 116.716,Z 834.311,A -85,B 0,C 180,E1 -26041.797,E2 -26041.797} C_VEL
LIN {X 0,Y 121.439,Z 827.519,A -85,B 0,C 180,E1 -26046.387,E2 -26046.387} C_VEL
LIN {X 0,Y 126.973,Z 819.032,A -85,B 0,C 180,E1 -26050.572,E2 -26050.572} C_VEL
LIN {X 0,Y 132.157,Z 810.308,A -85,B 0,C 180,E1 -26053.738,E2 -26053.738} C_VEL
LIN {X 0,Y 137.176,Z 800.732,A -85,B 0,C 180,E1 -26056.361,E2 -26056.361} C_VEL
LIN {X 0,Y 141.865,Z 790.255,A -85,B 0,C 180,E1 -26058.532,E2 -26058.532} C_VEL
LIN {X 0,Y 146.085,Z 778.546,A -85,B 0,C 180,E1 -26060.333,E2 -26060.333} C_VEL
LIN {X 0,Y 149.566,Z 766.442,A -85,B 0,C 180,E1 -26061.643,E2 -26061.643} C_VEL
LIN {X 0,Y 152.229,Z 753.897,A -85,B 0,C 180,E1 -26062.546,E2 -26062.546} C_VEL
LIN {X 0,Y 153.903,Z 739.082,A -85,B 0,C 180,E1 -26063.244,E2 -26063.244} C_VEL
LIN {X 0,Y 157.018,Z 699.41,A -85,B 0,C 180,E1 -26064.712,E2 -26064.712} C_VEL
LIN {X 0,Y 156.757,Z 676.251,A -85,B 0,C 180,E1 -26066.686,E2 -26066.686} C_VEL
LIN {X 0,Y 156.239,Z 661.755,A -85,B 0,C 180,E1 -26068.188,E2 -26068.188} C_VEL
LIN {X 0,Y 154.974,Z 657.467,A -85,B 0,C 180,E1 -26069.324,E2 -26069.324} C_VEL
LIN {X 0,Y 150.653,Z 650.159,A -85,B 0,C 180,E1 -26072.945,E2 -26072.945} C_VEL
LIN {X 0,Y 146.079,Z 643.142,A -85,B 0,C 180,E1 -26077.55,E2 -26077.55} C_VEL
LIN {X 0,Y 141.904,Z 637.456,A -85,B 0,C 180,E1 -26082.97,E2 -26082.97} C_VEL
LIN {X 0,Y 138.82,Z 633.684,A -85,B 0,C 180,E1 -26088.687,E2 -26088.687} C_VEL
LIN {X 0,Y 137.086,Z 631.554,A -85,B 0,C 180,E1 -26094.115,E2 -26094.115} C_VEL
LIN {X 0,Y 136.517,Z 630.534,A -85,B 0,C 180,E1 -26098.525,E2 -26098.525} C_VEL
LIN {X 0,Y 136.461,Z 630.647,A -85,B 0,C 180,E1 -26100.738,E2 -26100.738} C_VEL
LIN {X 0,Y 137.606,Z 633.13,A -85,B 0,C 180,E1 -26108.444,E2 -26108.444} C_VEL
LIN {X 0,Y 139.858,Z 636.754,A -85,B 0,C 180,E1 -26114.095,E2 -26114.095} C_VEL
LIN {X 0,Y 143.649,Z 642.777,A -85,B 0,C 180,E1 -26120.12,E2 -26120.12} C_VEL
LIN {X 0,Y 146.72,Z 648.171,A -85,B 0,C 180,E1 -26123.839,E2 -26123.839} C_VEL
LIN {X 0,Y 150.753,Z 655.747,A -85,B 0,C 180,E1 -26127.882,E2 -26127.882} C_VEL
LIN {X 0,Y 154.526,Z 663.861,A -85,B 0,C 180,E1 -26131.155,E2 -26131.155} C_VEL
LIN {X 0,Y 158.235,Z 673.193,A -85,B 0,C 180,E1 -26134.068,E2 -26134.068} C_VEL
LIN {X 0,Y 158.784,Z 675.098,A -85,B 0,C 180,E1 -26134.511,E2 -26134.511} C_VEL
LIN {X 0,Y 158.992,Z 680.664,A -85,B 0,C 180,E1 -26135.053,E2 -26135.053} C_VEL
LIN {X 0,Y 153.629,Z 743.41,A -85,B 0,C 180,E1 -26137.3,E2 -26137.3} C_VEL
LIN {X 0,Y 151.38,Z 756.533,A -85,B 0,C 180,E1 -26138.153,E2 -26138.153} C_VEL
LIN {X 0,Y 148.379,Z 768.872,A -85,B 0,C 180,E1 -26139.406,E2 -26139.406} C_VEL
LIN {X 0,Y 144.487,Z 780.78,A -85,B 0,C 180,E1 -26141.065,E2 -26141.065} C_VEL
LIN {X 0,Y 139.859,Z 792.063,A -85,B 0,C 180,E1 -26143.226,E2 -26143.226} C_VEL
LIN {X 0,Y 134.896,Z 802.247,A -85,B 0,C 180,E1 -26145.824,E2 -26145.824} C_VEL
LIN {X 0,Y 130.265,Z 810.578,A -85,B 0,C 180,E1 -26148.628,E2 -26148.628} C_VEL
LIN {X 0,Y 125.515,Z 818.248,A -85,B 0,C 180,E1 -26151.978,E2 -26151.978} C_VEL
LIN {X 0,Y 120.344,Z 825.722,A -85,B 0,C 180,E1 -26156.301,E2 -26156.301} C_VEL
LIN {X 0,Y 115.689,Z 831.725,A -85,B 0,C 180,E1 -26160.92,E2 -26160.92} C_VEL
LIN {X 0,Y 111.961,Z 836.46,A -85,B 0,C 180,E1 -26165.917,E2 -26165.917} C_VEL
LIN {X 0,Y 109.01,Z 840.076,A -85,B 0,C 180,E1 -26171.192,E2 -26171.192} C_VEL
LIN {X 0,Y 107.559,Z 841.935,A -85,B 0,C 180,E1 -26174.846,E2 -26174.846} C_VEL
LIN {X 0,Y 106.455,Z 843.349,A -85,B 0,C 180,E1 -26178.574,E2 -26178.574} C_VEL
LIN {X 0,Y 105.338,Z 844.948,A -85,B 0,C 180,E1 -26186.171,E2 -26186.171} C_VEL
LIN {X 0,Y 105.237,Z 845.176,A -85,B 0,C 180,E1 -26189.997,E2 -26189.997} C_VEL
LIN {X 0,Y 105.715,Z 844.388,A -85,B 0,C 180,E1 -26197.637,E2 -26197.637} C_VEL
LIN {X 0,Y 106.452,Z 843.416,A -85,B 0,C 180,E1 -26201.42,E2 -26201.42} C_VEL
LIN {X 0,Y 107.552,Z 842.041,A -85,B 0,C 180,E1 -26205.148,E2 -26205.148} C_VEL
LIN {X 0,Y 109.859,Z 839.152,A -85,B 0,C 180,E1 -26210.597,E2 -26210.597} C_VEL
LIN {X 0,Y 113.021,Z 835.221,A -85,B 0,C 180,E1 -26215.799,E2 -26215.799} C_VEL
LIN {X 0,Y 117.118,Z 830.123,A -85,B 0,C 180,E1 -26220.664,E2 -26220.664} C_VEL
LIN {X 0,Y 121.924,Z 823.696,A -85,B 0,C 180,E1 -26225.195,E2 -26225.195} C_VEL
LIN {X 0,Y 127.586,Z 815.231,A -85,B 0,C 180,E1 -26229.628,E2 -26229.628} C_VEL
LIN {X 0,Y 132.191,Z 807.5,A -85,B 0,C 180,E1 -26232.672,E2 -26232.672} C_VEL
LIN {X 0,Y 137.532,Z 797.392,A -85,B 0,C 180,E1 -26235.673,E2 -26235.673} C_VEL
LIN {X 0,Y 142.54,Z 786.381,A -85,B 0,C 180,E1 -26238.08,E2 -26238.08} C_VEL
LIN {X 0,Y 143.821,Z 783.116,A -85,B 0,C 180,E1 -26238.675,E2 -26238.675} C_VEL
LIN {X 0,Y 143.597,Z 781.192,A -85,B 0,C 180,E1 -26239.46,E2 -26239.46} C_VEL
LIN {X 0,Y 137.538,Z 782.252,A -85,B 0,C 180,E1 -26242.18,E2 -26242.18} C_VEL
LIN {X 0,Y 133.465,Z 782.165,A -85,B 0,C 180,E1 -26244.603,E2 -26244.603} C_VEL
LIN {X 0,Y 129.341,Z 782.711,A -85,B 0,C 180,E1 -26247.086,E2 -26247.086} C_VEL
LIN {X 0,Y 126.161,Z 781.865,A -85,B 0,C 180,E1 -26249.91,E2 -26249.91} C_VEL
LIN {X 0,Y 122.647,Z 782.314,A -85,B 0,C 180,E1 -26252.715,E2 -26252.715} C_VEL
LIN {X 0,Y 120.133,Z 781.421,A -85,B 0,C 180,E1 -26255.825,E2 -26255.825} C_VEL
LIN {X 0,Y 117.688,Z 781.059,A -85,B 0,C 180,E1 -26259.004,E2 -26259.004} C_VEL
LIN {X 0,Y 113.538,Z 778.26,A -85,B 0,C 180,E1 -26269.298,E2 -26269.298} C_VEL
LIN {X 0,Y 113.259,Z 776.629,A -85,B 0,C 180,E1 -26273.107,E2 -26273.107} C_VEL
LIN {X 0,Y 113.496,Z 775.86,A -85,B 0,C 180,E1 -26273.735,E2 -26273.735} C_VEL
LIN {X 0,Y 118.282,Z 779.663,A -85,B 0,C 180,E1 -26280,E2 -26280} C_VEL
LIN {X 0,Y 121.574,Z 781.196,A -85,B 0,C 180,E1 -26283.314,E2 -26283.314} C_VEL
LIN {X 0,Y 127.863,Z 782.728,A -85,B 0,C 180,E1 -26288.384,E2 -26288.384} C_VEL
LIN {X 0,Y 133.648,Z 783.119,A -85,B 0,C 180,E1 -26292.142,E2 -26292.142} C_VEL
LIN {X 0,Y 138.319,Z 782.883,A -85,B 0,C 180,E1 -26294.717,E2 -26294.717} C_VEL
LIN {X 0,Y 143.247,Z 782.222,A -85,B 0,C 180,E1 -26297.12,E2 -26297.12} C_VEL
LIN {X 0,Y 149.276,Z 780.936,A -85,B 0,C 180,E1 -26299.685,E2 -26299.685} C_VEL
LIN {X 0,Y 159.461,Z 777.538,A -85,B 0,C 180,E1 -26303.37,E2 -26303.37} C_VEL
LIN {X 0,Y 168.251,Z 773.549,A -85,B 0,C 180,E1 -26306.014,E2 -26306.014} C_VEL
LIN {X 0,Y 177.279,Z 768.364,A -85,B 0,C 180,E1 -26308.406,E2 -26308.406} C_VEL
LIN {X 0,Y 186.643,Z 761.808,A -85,B 0,C 180,E1 -26310.527,E2 -26310.527} C_VEL
LIN {X 0,Y 184.981,Z 763.494,A -85,B 0,C 180,E1 -26311.262,E2 -26311.262} C_VEL
LIN {X 0,Y 175.492,Z 771.329,A -85,B 0,C 180,E1 -26312.76,E2 -26312.76} C_VEL
LIN {X 0,Y 166.305,Z 777.977,A -85,B 0,C 180,E1 -26314.511,E2 -26314.511} C_VEL
LIN {X 0,Y 154.587,Z 785.14,A -85,B 0,C 180,E1 -26317.293,E2 -26317.293} C_VEL
LIN {X 0,Y 143.783,Z 790.746,A -85,B 0,C 180,E1 -26320.749,E2 -26320.749} C_VEL
LIN {X 0,Y 141.215,Z 792.085,A -85,B 0,C 180,E1 -26321.715,E2 -26321.715} C_VEL
LIN {X 0,Y 136.034,Z 803.388,A -85,B 0,C 180,E1 -26324.211,E2 -26324.211} C_VEL
LIN {X 0,Y 131.13,Z 812.498,A -85,B 0,C 180,E1 -26326.899,E2 -26326.899} C_VEL
LIN {X 0,Y 125.098,Z 822.287,A -85,B 0,C 180,E1 -26330.804,E2 -26330.804} C_VEL
LIN {X 0,Y 120.64,Z 828.935,A -85,B 0,C 180,E1 -26334.373,E2 -26334.373} C_VEL
LIN {X 0,Y 115.985,Z 835.466,A -85,B 0,C 180,E1 -26339.003,E2 -26339.003} C_VEL
LIN {X 0,Y 112.727,Z 839.653,A -85,B 0,C 180,E1 -26342.884,E2 -26342.884} C_VEL
LIN {X 0,Y 110.321,Z 841.985,A -85,B 0,C 180,E1 -26345.39,E2 -26345.39} C_VEL
LIN {X 0,Y 105.071,Z 845.167,A -85,B 0,C 180,E1 -26349.538,E2 -26349.538} C_VEL
LIN {X 0,Y 101.134,Z 847.19,A -85,B 0,C 180,E1 -26353.212,E2 -26353.212} C_VEL
LIN {X 0,Y 99.203,Z 848.427,A -85,B 0,C 180,E1 -26356.326,E2 -26356.326} C_VEL
LIN {X 0,Y 98.882,Z 848.771,A -85,B 0,C 180,E1 -26357.426,E2 -26357.426} C_VEL
LIN {X 0,Y 98.25,Z 849.87,A -85,B 0,C 180,E1 -26361.778,E2 -26361.778} C_VEL
LIN {X 0,Y 98.074,Z 850.489,A -85,B 0,C 180,E1 -26365.894,E2 -26365.894} C_VEL
LIN {X 0,Y 98.193,Z 850.708,A -85,B 0,C 180,E1 -26370.003,E2 -26370.003} C_VEL
LIN {X 0,Y 98.075,Z 850.471,A -85,B 0,C 180,E1 -26374.113,E2 -26374.113} C_VEL
LIN {X 0,Y 98.832,Z 848.819,A -85,B 0,C 180,E1 -26382.321,E2 -26382.321} C_VEL
LIN {X 0,Y 99.855,Z 847.373,A -85,B 0,C 180,E1 -26386.355,E2 -26386.355} C_VEL
LIN {X 0,Y 102.174,Z 844.385,A -85,B 0,C 180,E1 -26392.232,E2 -26392.232} C_VEL
LIN {X 0,Y 105.589,Z 840.343,A -85,B 0,C 180,E1 -26397.773,E2 -26397.773} C_VEL
LIN {X 0,Y 110.715,Z 834.117,A -85,B 0,C 180,E1 -26403.744,E2 -26403.744} C_VEL
LIN {X 0,Y 115.761,Z 827.326,A -85,B 0,C 180,E1 -26408.486,E2 -26408.486} C_VEL
LIN {X 0,Y 120.623,Z 820.399,A -85,B 0,C 180,E1 -26412.073,E2 -26412.073} C_VEL
LIN {X 0,Y 125.991,Z 812.041,A -85,B 0,C 180,E1 -26415.337,E2 -26415.337} C_VEL
LIN {X 0,Y 131.746,Z 801.7,A -85,B 0,C 180,E1 -26418.319,E2 -26418.319} C_VEL
LIN {X 0,Y 137.264,Z 790.071,A -85,B 0,C 180,E1 -26420.754,E2 -26420.754} C_VEL
LIN {X 0,Y 141.66,Z 778.368,A -85,B 0,C 180,E1 -26422.543,E2 -26422.543} C_VEL
LIN {X 0,Y 145.277,Z 766.273,A -85,B 0,C 180,E1 -26423.834,E2 -26423.834} C_VEL
LIN {X 0,Y 148.085,Z 753.327,A -85,B 0,C 180,E1 -26424.752,E2 -26424.752} C_VEL
LIN {X 0,Y 149.829,Z 738.348,A -85,B 0,C 180,E1 -26425.436,E2 -26425.436} C_VEL
LIN {X 0,Y 152.949,Z 700.436,A -85,B 0,C 180,E1 -26426.832,E2 -26426.832} C_VEL
LIN {X 0,Y 152.888,Z 677.308,A -85,B 0,C 180,E1 -26428.858,E2 -26428.858} C_VEL
LIN {X 0,Y 152.531,Z 664.631,A -85,B 0,C 180,E1 -26430.233,E2 -26430.233} C_VEL
LIN {X 0,Y 151.802,Z 662.295,A -85,B 0,C 180,E1 -26430.936,E2 -26430.936} C_VEL
LIN {X 0,Y 147.418,Z 654.725,A -85,B 0,C 180,E1 -26434.992,E2 -26434.992} C_VEL
LIN {X 0,Y 144.205,Z 649.47,A -85,B 0,C 180,E1 -26438.56,E2 -26438.56} C_VEL
LIN {X 0,Y 140.434,Z 644.096,A -85,B 0,C 180,E1 -26443.808,E2 -26443.808} C_VEL
LIN {X 0,Y 137.661,Z 640.504,A -85,B 0,C 180,E1 -26449.335,E2 -26449.335} C_VEL
LIN {X 0,Y 135.948,Z 638.23,A -85,B 0,C 180,E1 -26455.553,E2 -26455.553} C_VEL
LIN {X 0,Y 135.651,Z 637.588,A -85,B 0,C 180,E1 -26458.516,E2 -26458.516} C_VEL
LIN {X 0,Y 135.586,Z 637.771,A -85,B 0,C 180,E1 -26460.743,E2 -26460.743} C_VEL
LIN {X 0,Y 136.53,Z 639.969,A -85,B 0,C 180,E1 -26467.766,E2 -26467.766} C_VEL
LIN {X 0,Y 138.518,Z 643.414,A -85,B 0,C 180,E1 -26473.246,E2 -26473.246} C_VEL
LIN {X 0,Y 141.918,Z 649.186,A -85,B 0,C 180,E1 -26479.106,E2 -26479.106} C_VEL
LIN {X 0,Y 144.596,Z 654.216,A -85,B 0,C 180,E1 -26482.627,E2 -26482.627} C_VEL
LIN {X 0,Y 148.139,Z 661.279,A -85,B 0,C 180,E1 -26486.496,E2 -26486.496} C_VEL
LIN {X 0,Y 151.47,Z 668.895,A -85,B 0,C 180,E1 -26489.657,E2 -26489.657} C_VEL
LIN {X 0,Y 154.717,Z 677.505,A -85,B 0,C 180,E1 -26492.452,E2 -26492.452} C_VEL
LIN {X 0,Y 154.936,Z 679.945,A -85,B 0,C 180,E1 -26492.786,E2 -26492.786} C_VEL
LIN {X 0,Y 154.761,Z 683.791,A -85,B 0,C 180,E1 -26493.008,E2 -26493.008} C_VEL
LIN {X 0,Y 149.452,Z 743.533,A -85,B 0,C 180,E1 -26495.142,E2 -26495.142} C_VEL
LIN {X 0,Y 147.113,Z 756.698,A -85,B 0,C 180,E1 -26495.984,E2 -26495.984} C_VEL
LIN {X 0,Y 143.978,Z 769.048,A -85,B 0,C 180,E1 -26497.223,E2 -26497.223} C_VEL
LIN {X 0,Y 139.933,Z 780.962,A -85,B 0,C 180,E1 -26498.877,E2 -26498.877} C_VEL
LIN {X 0,Y 135.093,Z 792.25,A -85,B 0,C 180,E1 -26501.03,E2 -26501.03} C_VEL
LIN {X 0,Y 129.9,Z 802.435,A -85,B 0,C 180,E1 -26503.642,E2 -26503.642} C_VEL
LIN {X 0,Y 125.015,Z 810.769,A -85,B 0,C 180,E1 -26506.473,E2 -26506.473} C_VEL
LIN {X 0,Y 120.007,Z 818.439,A -85,B 0,C 180,E1 -26509.892,E2 -26509.892} C_VEL
LIN {X 0,Y 114.513,Z 825.914,A -85,B 0,C 180,E1 -26514.332,E2 -26514.332} C_VEL
LIN {X 0,Y 109.547,Z 831.917,A -85,B 0,C 180,E1 -26519.117,E2 -26519.117} C_VEL
LIN {X 0,Y 105.519,Z 836.653,A -85,B 0,C 180,E1 -26524.344,E2 -26524.344} C_VEL
LIN {X 0,Y 102.306,Z 840.269,A -85,B 0,C 180,E1 -26529.908,E2 -26529.908} C_VEL
LIN {X 0,Y 100.71,Z 842.129,A -85,B 0,C 180,E1 -26533.788,E2 -26533.788} C_VEL
LIN {X 0,Y 99.512,Z 843.542,A -85,B 0,C 180,E1 -26537.765,E2 -26537.765} C_VEL
LIN {X 0,Y 98.256,Z 845.141,A -85,B 0,C 180,E1 -26545.895,E2 -26545.895} C_VEL
LIN {X 0,Y 98.151,Z 845.368,A -85,B 0,C 180,E1 -26549.997,E2 -26549.997} C_VEL
LIN {X 0,Y 98.215,Z 845.17,A -85,B 0,C 180,E1 -26554.1,E2 -26554.1} C_VEL
LIN {X 0,Y 98.682,Z 844.581,A -85,B 0,C 180,E1 -26558.185,E2 -26558.185} C_VEL
LIN {X 0,Y 99.509,Z 843.609,A -85,B 0,C 180,E1 -26562.229,E2 -26562.229} C_VEL
LIN {X 0,Y 100.702,Z 842.233,A -85,B 0,C 180,E1 -26566.206,E2 -26566.206} C_VEL
LIN {X 0,Y 103.249,Z 839.344,A -85,B 0,C 180,E1 -26571.982,E2 -26571.982} C_VEL
LIN {X 0,Y 106.657,Z 835.413,A -85,B 0,C 180,E1 -26577.464,E2 -26577.464} C_VEL
LIN {X 0,Y 111.078,Z 830.312,A -85,B 0,C 180,E1 -26582.53,E2 -26582.53} C_VEL
LIN {X 0,Y 116.19,Z 823.884,A -85,B 0,C 180,E1 -26587.215,E2 -26587.215} C_VEL
LIN {X 0,Y 121.279,Z 816.76,A -85,B 0,C 180,E1 -26591.119,E2 -26591.119} C_VEL
LIN {X 0,Y 127.07,Z 807.684,A -85,B 0,C 180,E1 -26594.839,E2 -26594.839} C_VEL
LIN {X 0,Y 132.673,Z 797.572,A -85,B 0,C 180,E1 -26597.864,E2 -26597.864} C_VEL
LIN {X 0,Y 136.759,Z 789.198,A -85,B 0,C 180,E1 -26599.755,E2 -26599.755} C_VEL
LIN {X 0,Y 136.935,Z 787.976,A -85,B 0,C 180,E1 -26600.177,E2 -26600.177} C_VEL
LIN {X 0,Y 134.677,Z 788.325,A -85,B 0,C 180,E1 -26601.229,E2 -26601.229} C_VEL
LIN {X 0,Y 130.511,Z 788.264,A -85,B 0,C 180,E1 -26603.676,E2 -26603.676} C_VEL
LIN {X 0,Y 126.291,Z 788.789,A -85,B 0,C 180,E1 -26606.186,E2 -26606.186} C_VEL
LIN {X 0,Y 123.029,Z 788.02,A -85,B 0,C 180,E1 -26609.061,E2 -26609.061} C_VEL
LIN {X 0,Y 119.102,Z 788.389,A -85,B 0,C 180,E1 -26612.259,E2 -26612.259} C_VEL
LIN {X 0,Y 116.864,Z 787.608,A -85,B 0,C 180,E1 -26615.104,E2 -26615.104} C_VEL
LIN {X 0,Y 114.402,Z 787.237,A -85,B 0,C 180,E1 -26618.371,E2 -26618.371} C_VEL
LIN {X 0,Y 110.216,Z 784.61,A -85,B 0,C 180,E1 -26628.971,E2 -26628.971} C_VEL
LIN {X 0,Y 109.935,Z 782.222,A -85,B 0,C 180,E1 -26636.334,E2 -26636.334} C_VEL
LIN {X 0,Y 110.916,Z 780.049,A -85,B 0,C 180,E1 -26640.348,E2 -26640.348} C_VEL
LIN {X 0,Y 111.175,Z 779.771,A -85,B 0,C 180,E1 -26640.695,E2 -26640.695} C_VEL
LIN {X 0,Y 117.628,Z 782.694,A -85,B 0,C 180,E1 -26646.863,E2 -26646.863} C_VEL
LIN {X 0,Y 121.749,Z 783.699,A -85,B 0,C 180,E1 -26649.972,E2 -26649.972} C_VEL
LIN {X 0,Y 126.193,Z 784.293,A -85,B 0,C 180,E1 -26652.872,E2 -26652.872} C_VEL
LIN {X 0,Y 131.491,Z 784.429,A -85,B 0,C 180,E1 -26655.843,E2 -26655.843} C_VEL
LIN {X 0,Y 141.377,Z 783.432,A -85,B 0,C 180,E1 -26660.364,E2 -26660.364} C_VEL
LIN {X 0,Y 146.961,Z 782.295,A -85,B 0,C 180,E1 -26662.493,E2 -26662.493} C_VEL
LIN {X 0,Y 155.537,Z 779.755,A -85,B 0,C 180,E1 -26665.357,E2 -26665.357} C_VEL
LIN {X 0,Y 164.792,Z 775.974,A -85,B 0,C 180,E1 -26667.977,E2 -26667.977} C_VEL
LIN {X 0,Y 173.51,Z 771.529,A -85,B 0,C 180,E1 -26670.121,E2 -26670.121} C_VEL
LIN {X 0,Y 172.804,Z 772.192,A -85,B 0,C 180,E1 -26670.618,E2 -26670.618} C_VEL
LIN {X 0,Y 162.41,Z 778.98,A -85,B 0,C 180,E1 -26672.459,E2 -26672.459} C_VEL
LIN {X 0,Y 150.402,Z 785.592,A -85,B 0,C 180,E1 -26675.146,E2 -26675.146} C_VEL
LIN {X 0,Y 139.25,Z 790.673,A -85,B 0,C 180,E1 -26678.534,E2 -26678.534} C_VEL
LIN {X 0,Y 136.6,Z 791.91,A -85,B 0,C 180,E1 -26679.494,E2 -26679.494} C_VEL
LIN {X 0,Y 131.179,Z 803.207,A -85,B 0,C 180,E1 -26681.986,E2 -26681.986} C_VEL
LIN {X 0,Y 126.038,Z 812.314,A -85,B 0,C 180,E1 -26684.692,E2 -26684.692} C_VEL
LIN {X 0,Y 119.651,Z 822.1,A -85,B 0,C 180,E1 -26688.644,E2 -26688.644} C_VEL
LIN {X 0,Y 113.967,Z 830.042,A -85,B 0,C 180,E1 -26693.12,E2 -26693.12} C_VEL
LIN {X 0,Y 109.955,Z 835.277,A -85,B 0,C 180,E1 -26697.096,E2 -26697.096} C_VEL
LIN {X 0,Y 105.629,Z 840.463,A -85,B 0,C 180,E1 -26702.246,E2 -26702.246} C_VEL
LIN {X 0,Y 102.195,Z 844.477,A -85,B 0,C 180,E1 -26707.779,E2 -26707.779} C_VEL
LIN {X 0,Y 99.859,Z 847.441,A -85,B 0,C 180,E1 -26713.653,E2 -26713.653} C_VEL
LIN {X 0,Y 98.882,Z 848.771,A -85,B 0,C 180,E1 -26717.426,E2 -26717.426} C_VEL
LIN {X 0,Y 97.689,Z 849.743,A -85,B 0,C 180,E1 -26720.756,E2 -26720.756} C_VEL
LIN {X 0,Y 95.818,Z 850.341,A -85,B 0,C 180,E1 -26724.085,E2 -26724.085} C_VEL
LIN {X 0,Y 91.997,Z 850.542,A -85,B 0,C 180,E1 -26731.063,E2 -26731.063} C_VEL
LIN {X 0,Y 91.004,Z 850.048,A -85,B 0,C 180,E1 -26736.046,E2 -26736.046} C_VEL
LIN {X 0,Y 91.881,Z 848.625,A -85,B 0,C 180,E1 -26743.27,E2 -26743.27} C_VEL
LIN {X 0,Y 93.024,Z 847.179,A -85,B 0,C 180,E1 -26747.593,E2 -26747.593} C_VEL
LIN {X 0,Y 95.6,Z 844.19,A -85,B 0,C 180,E1 -26753.853,E2 -26753.853} C_VEL
LIN {X 0,Y 99.316,Z 840.148,A -85,B 0,C 180,E1 -26759.696,E2 -26759.696} C_VEL
LIN {X 0,Y 104.858,Z 833.924,A -85,B 0,C 180,E1 -26765.91,E2 -26765.91} C_VEL
LIN {X 0,Y 110.26,Z 827.134,A -85,B 0,C 180,E1 -26770.797,E2 -26770.797} C_VEL
LIN {X 0,Y 115.428,Z 820.207,A -85,B 0,C 180,E1 -26774.446,E2 -26774.446} C_VEL
LIN {X 0,Y 121.089,Z 811.851,A -85,B 0,C 180,E1 -26777.735,E2 -26777.735} C_VEL
LIN {X 0,Y 127.13,Z 801.513,A -85,B 0,C 180,E1 -26780.713,E2 -26780.713} C_VEL
LIN {X 0,Y 132.236,Z 791.294,A -85,B 0,C 180,E1 -26782.867,E2 -26782.867} C_VEL
LIN {X 0,Y 136.791,Z 780.102,A -85,B 0,C 180,E1 -26784.651,E2 -26784.651} C_VEL
LIN {X 0,Y 140.868,Z 767.361,A -85,B 0,C 180,E1 -26786.043,E2 -26786.043} C_VEL
LIN {X 0,Y 143.87,Z 754.476,A -85,B 0,C 180,E1 -26786.981,E2 -26786.981} C_VEL
LIN {X 0,Y 145.688,Z 740.756,A -85,B 0,C 180,E1 -26787.644,E2 -26787.644} C_VEL
LIN {X 0,Y 149.109,Z 701.338,A -85,B 0,C 180,E1 -26789.07,E2 -26789.07} C_VEL
LIN {X 0,Y 149.25,Z 678.911,A -85,B 0,C 180,E1 -26791.087,E2 -26791.087} C_VEL
LIN {X 0,Y 149.046,Z 667.695,A -85,B 0,C 180,E1 -26792.344,E2 -26792.344} C_VEL
LIN {X 0,Y 145.362,Z 661.011,A -85,B 0,C 180,E1 -26796.025,E2 -26796.025} C_VEL
LIN {X 0,Y 142.241,Z 655.65,A -85,B 0,C 180,E1 -26799.766,E2 -26799.766} C_VEL
LIN {X 0,Y 139.018,Z 650.767,A -85,B 0,C 180,E1 -26804.623,E2 -26804.623} C_VEL
LIN {X 0,Y 136.418,Z 647.215,A -85,B 0,C 180,E1 -26810.268,E2 -26810.268} C_VEL
LIN {X 0,Y 134.897,Z 644.901,A -85,B 0,C 180,E1 -26817.014,E2 -26817.014} C_VEL
LIN {X 0,Y 134.721,Z 644.763,A -85,B 0,C 180,E1 -26820.374,E2 -26820.374} C_VEL
LIN {X 0,Y 135.561,Z 646.991,A -85,B 0,C 180,E1 -26827.447,E2 -26827.447} C_VEL
LIN {X 0,Y 137.342,Z 650.34,A -85,B 0,C 180,E1 -26832.696,E2 -26832.696} C_VEL
LIN {X 0,Y 140.285,Z 655.708,A -85,B 0,C 180,E1 -26838.153,E2 -26838.153} C_VEL
LIN {X 0,Y 142.659,Z 660.517,A -85,B 0,C 180,E1 -26841.538,E2 -26841.538} C_VEL
LIN {X 0,Y 145.776,Z 667.17,A -85,B 0,C 180,E1 -26845.237,E2 -26845.237} C_VEL
LIN {X 0,Y 148.818,Z 674.727,A -85,B 0,C 180,E1 -26848.392,E2 -26848.392} C_VEL
LIN {X 0,Y 151.11,Z 681.158,A -85,B 0,C 180,E1 -26850.562,E2 -26850.562} C_VEL
LIN {X 0,Y 150.964,Z 684.433,A -85,B 0,C 180,E1 -26850.769,E2 -26850.769} C_VEL
LIN {X 0,Y 145.476,Z 743.803,A -85,B 0,C 180,E1 -26852.869,E2 -26852.869} C_VEL
LIN {X 0,Y 143.064,Z 756.863,A -85,B 0,C 180,E1 -26853.687,E2 -26853.687} C_VEL
LIN {X 0,Y 139.806,Z 769.223,A -85,B 0,C 180,E1 -26854.91,E2 -26854.91} C_VEL
LIN {X 0,Y 135.602,Z 781.144,A -85,B 0,C 180,E1 -26856.547,E2 -26856.547} C_VEL
LIN {X 0,Y 130.556,Z 792.436,A -85,B 0,C 180,E1 -26858.685,E2 -26858.685} C_VEL
LIN {X 0,Y 125.109,Z 802.624,A -85,B 0,C 180,E1 -26861.29,E2 -26861.29} C_VEL
LIN {X 0,Y 119.973,Z 810.959,A -85,B 0,C 180,E1 -26864.14,E2 -26864.14} C_VEL
LIN {X 0,Y 114.673,Z 818.631,A -85,B 0,C 180,E1 -26867.608,E2 -26867.608} C_VEL
LIN {X 0,Y 108.831,Z 826.106,A -85,B 0,C 180,E1 -26872.155,E2 -26872.155} C_VEL
LIN {X 0,Y 103.528,Z 832.11,A -85,B 0,C 180,E1 -26877.103,E2 -26877.103} C_VEL
LIN {X 0,Y 99.144,Z 836.847,A -85,B 0,C 180,E1 -26882.56,E2 -26882.56} C_VEL
LIN {X 0,Y 95.669,Z 840.463,A -85,B 0,C 180,E1 -26888.447,E2 -26888.447} C_VEL
LIN {X 0,Y 93.91,Z 842.322,A -85,B 0,C 180,E1 -26892.578,E2 -26892.578} C_VEL
LIN {X 0,Y 92.58,Z 843.735,A -85,B 0,C 180,E1 -26896.833,E2 -26896.833} C_VEL
LIN {X 0,Y 91.679,Z 844.726,A -85,B 0,C 180,E1 -26901.177,E2 -26901.177} C_VEL
LIN {X 0,Y 91.183,Z 845.334,A -85,B 0,C 180,E1 -26905.576,E2 -26905.576} C_VEL
LIN {X 0,Y 91.056,Z 845.561,A -85,B 0,C 180,E1 -26909.996,E2 -26909.996} C_VEL
LIN {X 0,Y 91.677,Z 844.773,A -85,B 0,C 180,E1 -26918.816,E2 -26918.816} C_VEL
LIN {X 0,Y 92.577,Z 843.801,A -85,B 0,C 180,E1 -26923.16,E2 -26923.16} C_VEL
LIN {X 0,Y 93.902,Z 842.425,A -85,B 0,C 180,E1 -26927.416,E2 -26927.416} C_VEL
LIN {X 0,Y 96.691,Z 839.535,A -85,B 0,C 180,E1 -26933.559,E2 -26933.559} C_VEL
LIN {X 0,Y 100.398,Z 835.604,A -85,B 0,C 180,E1 -26939.337,E2 -26939.337} C_VEL
LIN {X 0,Y 105.158,Z 830.502,A -85,B 0,C 180,E1 -26944.612,E2 -26944.612} C_VEL
LIN {X 0,Y 110.613,Z 824.072,A -85,B 0,C 180,E1 -26949.442,E2 -26949.442} C_VEL
LIN {X 0,Y 116.65,Z 816.07,A -85,B 0,C 180,E1 -26953.85,E2 -26953.85} C_VEL
LIN {X 0,Y 122.135,Z 807.868,A -85,B 0,C 180,E1 -26957.19,E2 -26957.19} C_VEL
LIN {X 0,Y 128.019,Z 797.752,A -85,B 0,C 180,E1 -26960.221,E2 -26960.221} C_VEL
LIN {X 0,Y 129.268,Z 795.461,A -85,B 0,C 180,E1 -26960.776,E2 -26960.776} C_VEL
LIN {X 0,Y 128.703,Z 794.168,A -85,B 0,C 180,E1 -26961.789,E2 -26961.789} C_VEL
LIN {X 0,Y 123.004,Z 794.658,A -85,B 0,C 180,E1 -26965.154,E2 -26965.154} C_VEL
LIN {X 0,Y 119.631,Z 793.986,A -85,B 0,C 180,E1 -26968.08,E2 -26968.08} C_VEL
LIN {X 0,Y 115.974,Z 794.316,A -85,B 0,C 180,E1 -26971,E2 -26971} C_VEL
LIN {X 0,Y 108.918,Z 792.461,A -85,B 0,C 180,E1 -26981.178,E2 -26981.178} C_VEL
LIN {X 0,Y 106.572,Z 790.74,A -85,B 0,C 180,E1 -26988.589,E2 -26988.589} C_VEL
LIN {X 0,Y 106.354,Z 788.463,A -85,B 0,C 180,E1 -26996.211,E2 -26996.211} C_VEL
LIN {X 0,Y 108.208,Z 785.647,A -85,B 0,C 180,E1 -27003.724,E2 -27003.724} C_VEL
LIN {X 0,Y 110.486,Z 783.201,A -85,B 0,C 180,E1 -27007.768,E2 -27007.768} C_VEL
LIN {X 0,Y 118.748,Z 785.144,A -85,B 0,C 180,E1 -27013.694,E2 -27013.694} C_VEL
LIN {X 0,Y 125.131,Z 785.734,A -85,B 0,C 180,E1 -27017.303,E2 -27017.303} C_VEL
LIN {X 0,Y 134.332,Z 785.421,A -85,B 0,C 180,E1 -27021.483,E2 -27021.483} C_VEL
LIN {X 0,Y 140.037,Z 784.686,A -85,B 0,C 180,E1 -27023.672,E2 -27023.672} C_VEL
LIN {X 0,Y 149.598,Z 782.523,A -85,B 0,C 180,E1 -27026.804,E2 -27026.804} C_VEL
LIN {X 0,Y 159.588,Z 779.18,A -85,B 0,C 180,E1 -27029.53,E2 -27029.53} C_VEL
LIN {X 0,Y 157.684,Z 780.453,A -85,B 0,C 180,E1 -27030.489,E2 -27030.489} C_VEL
LIN {X 0,Y 146.44,Z 785.918,A -85,B 0,C 180,E1 -27032.88,E2 -27032.88} C_VEL
LIN {X 0,Y 134.944,Z 790.529,A -85,B 0,C 180,E1 -27036.177,E2 -27036.177} C_VEL
LIN {X 0,Y 132.394,Z 791.449,A -85,B 0,C 180,E1 -27037.074,E2 -27037.074} C_VEL
LIN {X 0,Y 126.538,Z 803.027,A -85,B 0,C 180,E1 -27039.595,E2 -27039.595} C_VEL
LIN {X 0,Y 121.134,Z 812.13,A -85,B 0,C 180,E1 -27042.296,E2 -27042.296} C_VEL
LIN {X 0,Y 114.41,Z 821.913,A -85,B 0,C 180,E1 -27046.29,E2 -27046.29} C_VEL
LIN {X 0,Y 108.556,Z 829.607,A -85,B 0,C 180,E1 -27050.697,E2 -27050.697} C_VEL
LIN {X 0,Y 104.047,Z 835.086,A -85,B 0,C 180,E1 -27054.965,E2 -27054.965} C_VEL
LIN {X 0,Y 99.366,Z 840.272,A -85,B 0,C 180,E1 -27060.328,E2 -27060.328} C_VEL
LIN {X 0,Y 95.622,Z 844.284,A -85,B 0,C 180,E1 -27066.161,E2 -27066.161} C_VEL
LIN {X 0,Y 93.03,Z 847.248,A -85,B 0,C 180,E1 -27072.415,E2 -27072.415} C_VEL
LIN {X 0,Y 91.847,Z 848.704,A -85,B 0,C 180,E1 -27076.889,E2 -27076.889} C_VEL
LIN {X 0,Y 90.992,Z 850.296,A -85,B 0,C 180,E1 -27085.574,E2 -27085.574} C_VEL
LIN {X 0,Y 91.111,Z 850.516,A -85,B 0,C 180,E1 -27090.004,E2 -27090.004} C_VEL
LIN {X 0,Y 91.004,Z 850.048,A -85,B 0,C 180,E1 -27096.046,E2 -27096.046} C_VEL
LIN {X 0,Y 90.6,Z 849.478,A -85,B 0,C 180,E1 -27099.753,E2 -27099.753} C_VEL
LIN {X 0,Y 88.862,Z 847.951,A -85,B 0,C 180,E1 -27105.935,E2 -27105.935} C_VEL
LIN {X 0,Y 88.091,Z 845.734,A -85,B 0,C 180,E1 -27112.198,E2 -27112.198} C_VEL
LIN {X 0,Y 89.166,Z 843.952,A -85,B 0,C 180,E1 -27115.783,E2 -27115.783} C_VEL
LIN {X 0,Y 93.174,Z 839.954,A -85,B 0,C 180,E1 -27121.874,E2 -27121.874} C_VEL
LIN {X 0,Y 99.163,Z 833.73,A -85,B 0,C 180,E1 -27128.33,E2 -27128.33} C_VEL
LIN {X 0,Y 104.976,Z 826.941,A -85,B 0,C 180,E1 -27133.335,E2 -27133.335} C_VEL
LIN {X 0,Y 110.465,Z 820.016,A -85,B 0,C 180,E1 -27137.028,E2 -27137.028} C_VEL
LIN {X 0,Y 116.425,Z 811.661,A -85,B 0,C 180,E1 -27140.326,E2 -27140.326} C_VEL
LIN {X 0,Y 122.752,Z 801.326,A -85,B 0,C 180,E1 -27143.282,E2 -27143.282} C_VEL
LIN {X 0,Y 128.726,Z 789.703,A -85,B 0,C 180,E1 -27145.67,E2 -27145.67} C_VEL
LIN {X 0,Y 133.51,Z 778.012,A -85,B 0,C 180,E1 -27147.381,E2 -27147.381} C_VEL
LIN {X 0,Y 137.385,Z 765.932,A -85,B 0,C 180,E1 -27148.615,E2 -27148.615} C_VEL
LIN {X 0,Y 140.194,Z 753.975,A -85,B 0,C 180,E1 -27149.44,E2 -27149.44} C_VEL
LIN {X 0,Y 142.076,Z 740.156,A -85,B 0,C 180,E1 -27150.073,E2 -27150.073} C_VEL
LIN {X 0,Y 145.537,Z 701.448,A -85,B 0,C 180,E1 -27151.483,E2 -27151.483} C_VEL
LIN {X 0,Y 145.863,Z 678.509,A -85,B 0,C 180,E1 -27153.629,E2 -27153.629} C_VEL
LIN {X 0,Y 145.78,Z 671.896,A -85,B 0,C 180,E1 -27154.421,E2 -27154.421} C_VEL
LIN {X 0,Y 143.057,Z 666.827,A -85,B 0,C 180,E1 -27157.43,E2 -27157.43} C_VEL
LIN {X 0,Y 140.584,Z 662.181,A -85,B 0,C 180,E1 -27160.668,E2 -27160.668} C_VEL
LIN {X 0,Y 137.565,Z 657.344,A -85,B 0,C 180,E1 -27165.578,E2 -27165.578} C_VEL
LIN {X 0,Y 135.27,Z 654.025,A -85,B 0,C 180,E1 -27171.033,E2 -27171.033} C_VEL
LIN {X 0,Y 133.968,Z 651.8,A -85,B 0,C 180,E1 -27177.745,E2 -27177.745} C_VEL
LIN {X 0,Y 133.849,Z 651.929,A -85,B 0,C 180,E1 -27180.752,E2 -27180.752} C_VEL
LIN {X 0,Y 134.584,Z 653.989,A -85,B 0,C 180,E1 -27187.076,E2 -27187.076} C_VEL
LIN {X 0,Y 136.096,Z 657.07,A -85,B 0,C 180,E1 -27191.921,E2 -27191.921} C_VEL
LIN {X 0,Y 138.669,Z 662.162,A -85,B 0,C 180,E1 -27197.133,E2 -27197.133} C_VEL
LIN {X 0,Y 140.739,Z 666.718,A -85,B 0,C 180,E1 -27200.365,E2 -27200.365} C_VEL
LIN {X 0,Y 143.341,Z 672.719,A -85,B 0,C 180,E1 -27203.764,E2 -27203.764} C_VEL
LIN {X 0,Y 145.865,Z 679.421,A -85,B 0,C 180,E1 -27206.666,E2 -27206.666} C_VEL
LIN {X 0,Y 147.473,Z 684.131,A -85,B 0,C 180,E1 -27208.369,E2 -27208.369} C_VEL
LIN {X 0,Y 141.834,Z 743.385,A -85,B 0,C 180,E1 -27210.444,E2 -27210.444} C_VEL
LIN {X 0,Y 139.437,Z 756.305,A -85,B 0,C 180,E1 -27211.208,E2 -27211.208} C_VEL
LIN {X 0,Y 135.881,Z 769.397,A -85,B 0,C 180,E1 -27212.463,E2 -27212.463} C_VEL
LIN {X 0,Y 132.172,Z 779.666,A -85,B 0,C 180,E1 -27213.813,E2 -27213.813} C_VEL
LIN {X 0,Y 127.584,Z 790.071,A -85,B 0,C 180,E1 -27215.655,E2 -27215.655} C_VEL
LIN {X 0,Y 121.782,Z 800.722,A -85,B 0,C 180,E1 -27218.156,E2 -27218.156} C_VEL
LIN {X 0,Y 115.136,Z 811.149,A -85,B 0,C 180,E1 -27221.601,E2 -27221.601} C_VEL
LIN {X 0,Y 109.52,Z 818.823,A -85,B 0,C 180,E1 -27225.096,E2 -27225.096} C_VEL
LIN {X 0,Y 103.324,Z 826.298,A -85,B 0,C 180,E1 -27229.742,E2 -27229.742} C_VEL
LIN {X 0,Y 97.656,Z 832.302,A -85,B 0,C 180,E1 -27234.845,E2 -27234.845} C_VEL
LIN {X 0,Y 92.886,Z 837.041,A -85,B 0,C 180,E1 -27240.537,E2 -27240.537} C_VEL
LIN {X 0,Y 89.109,Z 840.656,A -85,B 0,C 180,E1 -27246.771,E2 -27246.771} C_VEL
LIN {X 0,Y 87.168,Z 842.515,A -85,B 0,C 180,E1 -27251.182,E2 -27251.182} C_VEL
LIN {X 0,Y 85.671,Z 843.929,A -85,B 0,C 180,E1 -27255.749,E2 -27255.749} C_VEL
LIN {X 0,Y 84.67,Z 844.919,A -85,B 0,C 180,E1 -27260.44,E2 -27260.44} C_VEL
LIN {X 0,Y 84.105,Z 845.527,A -85,B 0,C 180,E1 -27265.203,E2 -27265.203} C_VEL
LIN {X 0,Y 83.957,Z 845.754,A -85,B 0,C 180,E1 -27269.996,E2 -27269.996} C_VEL
LIN {X 0,Y 84.072,Z 845.556,A -85,B 0,C 180,E1 -27274.791,E2 -27274.791} C_VEL
LIN {X 0,Y 84.668,Z 844.965,A -85,B 0,C 180,E1 -27279.552,E2 -27279.552} C_VEL
LIN {X 0,Y 85.667,Z 843.994,A -85,B 0,C 180,E1 -27284.244,E2 -27284.244} C_VEL
LIN {X 0,Y 87.159,Z 842.617,A -85,B 0,C 180,E1 -27288.812,E2 -27288.812} C_VEL
LIN {X 0,Y 90.223,Z 839.727,A -85,B 0,C 180,E1 -27295.363,E2 -27295.363} C_VEL
LIN {X 0,Y 94.259,Z 835.795,A -85,B 0,C 180,E1 -27301.457,E2 -27301.457} C_VEL
LIN {X 0,Y 99.387,Z 830.692,A -85,B 0,C 180,E1 -27306.941,E2 -27306.941} C_VEL
LIN {X 0,Y 105.216,Z 824.261,A -85,B 0,C 180,E1 -27311.905,E2 -27311.905} C_VEL
LIN {X 0,Y 111.634,Z 816.257,A -85,B 0,C 180,E1 -27316.377,E2 -27316.377} C_VEL
LIN {X 0,Y 117.419,Z 808.052,A -85,B 0,C 180,E1 -27319.736,E2 -27319.736} C_VEL
LIN {X 0,Y 121.684,Z 801.286,A -85,B 0,C 180,E1 -27321.832,E2 -27321.832} C_VEL
LIN {X 0,Y 121.892,Z 800.025,A -85,B 0,C 180,E1 -27322.535,E2 -27322.535} C_VEL
LIN {X 0,Y 119.486,Z 800.264,A -85,B 0,C 180,E1 -27323.971,E2 -27323.971} C_VEL
LIN {X 0,Y 116.009,Z 799.698,A -85,B 0,C 180,E1 -27326.959,E2 -27326.959} C_VEL
LIN {X 0,Y 112.266,Z 799.972,A -85,B 0,C 180,E1 -27329.946,E2 -27329.946} C_VEL
LIN {X 0,Y 104.956,Z 798.266,A -85,B 0,C 180,E1 -27340.439,E2 -27340.439} C_VEL
LIN {X 0,Y 102.59,Z 796.655,A -85,B 0,C 180,E1 -27348.14,E2 -27348.14} C_VEL
LIN {X 0,Y 102.401,Z 794.508,A -85,B 0,C 180,E1 -27356.064,E2 -27356.064} C_VEL
LIN {X 0,Y 104.448,Z 791.841,A -85,B 0,C 180,E1 -27363.858,E2 -27363.858} C_VEL
LIN {X 0,Y 109.49,Z 788.024,A -85,B 0,C 180,E1 -27372.584,E2 -27372.584} C_VEL
LIN {X 0,Y 112.201,Z 785.889,A -85,B 0,C 180,E1 -27375.206,E2 -27375.206} C_VEL
LIN {X 0,Y 121.605,Z 787.059,A -85,B 0,C 180,E1 -27380.289,E2 -27380.289} C_VEL
LIN {X 0,Y 133.092,Z 786.734,A -85,B 0,C 180,E1 -27384.989,E2 -27384.989} C_VEL
LIN {X 0,Y 143.822,Z 785.056,A -85,B 0,C 180,E1 -27388.414,E2 -27388.414} C_VEL
LIN {X 0,Y 146.489,Z 784.423,A -85,B 0,C 180,E1 -27389.174,E2 -27389.174} C_VEL
LIN {X 0,Y 145.818,Z 784.892,A -85,B 0,C 180,E1 -27389.832,E2 -27389.832} C_VEL
LIN {X 0,Y 133.754,Z 789.353,A -85,B 0,C 180,E1 -27392.791,E2 -27392.791} C_VEL
LIN {X 0,Y 128.248,Z 791.21,A -85,B 0,C 180,E1 -27394.548,E2 -27394.548} C_VEL
LIN {X 0,Y 122.118,Z 802.846,A -85,B 0,C 180,E1 -27397.017,E2 -27397.017} C_VEL
LIN {X 0,Y 116.458,Z 811.945,A -85,B 0,C 180,E1 -27399.702,E2 -27399.702} C_VEL
LIN {X 0,Y 109.37,Z 821.726,A -85,B 0,C 180,E1 -27403.71,E2 -27403.71} C_VEL
LIN {X 0,Y 102.883,Z 829.699,A -85,B 0,C 180,E1 -27408.375,E2 -27408.375} C_VEL
LIN {X 0,Y 96.488,Z 836.743,A -85,B 0,C 180,E1 -27414.364,E2 -27414.364} C_VEL
LIN {X 0,Y 91.765,Z 841.517,A -85,B 0,C 180,E1 -27420.149,E2 -27420.149} C_VEL
LIN {X 0,Y 88.02,Z 845.167,A -85,B 0,C 180,E1 -27426.475,E2 -27426.475} C_VEL
LIN {X 0,Y 86.259,Z 847.055,A -85,B 0,C 180,E1 -27430.984,E2 -27430.984} C_VEL
LIN {X 0,Y 84.967,Z 848.476,A -85,B 0,C 180,E1 -27435.637,E2 -27435.637} C_VEL
LIN {X 0,Y 83.903,Z 850.103,A -85,B 0,C 180,E1 -27445.199,E2 -27445.199} C_VEL
LIN {X 0,Y 84.016,Z 850.323,A -85,B 0,C 180,E1 -27450.004,E2 -27450.004} C_VEL
LIN {X 0,Y 83.919,Z 849.912,A -85,B 0,C 180,E1 -27456.124,E2 -27456.124} C_VEL
LIN {X 0,Y 84.968,Z 848.431,A -85,B 0,C 180,E1 -27464.371,E2 -27464.371} C_VEL
LIN {X 0,Y 86.253,Z 846.984,A -85,B 0,C 180,E1 -27469.025,E2 -27469.025} C_VEL
LIN {X 0,Y 89.166,Z 843.952,A -85,B 0,C 180,E1 -27475.783,E2 -27475.783} C_VEL
LIN {X 0,Y 90.555,Z 841.986,A -85,B 0,C 180,E1 -27479.219,E2 -27479.219} C_VEL
LIN {X 0,Y 91.77,Z 838.299,A -85,B 0,C 180,E1 -27484.977,E2 -27484.977} C_VEL
LIN {X 0,Y 93.673,Z 834.022,A -85,B 0,C 180,E1 -27490.399,E2 -27490.399} C_VEL
LIN {X 0,Y 96.014,Z 831.028,A -85,B 0,C 180,E1 -27493.145,E2 -27493.145} C_VEL
LIN {X 0,Y 102.168,Z 824.114,A -85,B 0,C 180,E1 -27497.691,E2 -27497.691} C_VEL
LIN {X 0,Y 108.214,Z 816.658,A -85,B 0,C 180,E1 -27501.204,E2 -27501.204} C_VEL
LIN {X 0,Y 114.658,Z 807.622,A -85,B 0,C 180,E1 -27504.311,E2 -27504.311} C_VEL
LIN {X 0,Y 120.689,Z 797.569,A -85,B 0,C 180,E1 -27506.837,E2 -27506.837} C_VEL
LIN {X 0,Y 126.263,Z 786.439,A -85,B 0,C 180,E1 -27508.852,E2 -27508.852} C_VEL
LIN {X 0,Y 130.891,Z 774.927,A -85,B 0,C 180,E1 -27510.365,E2 -27510.365} C_VEL
LIN {X 0,Y 134.742,Z 762.387,A -85,B 0,C 180,E1 -27511.472,E2 -27511.472} C_VEL
LIN {X 0,Y 137.486,Z 749.478,A -85,B 0,C 180,E1 -27512.215,E2 -27512.215} C_VEL
LIN {X 0,Y 139.641,Z 729.632,A -85,B 0,C 180,E1 -27512.993,E2 -27512.993} C_VEL
LIN {X 0,Y 142.198,Z 702.336,A -85,B 0,C 180,E1 -27513.954,E2 -27513.954} C_VEL
LIN {X 0,Y 142.785,Z 678.325,A -85,B 0,C 180,E1 -27516.252,E2 -27516.252} C_VEL
LIN {X 0,Y 142.681,Z 676.214,A -85,B 0,C 180,E1 -27516.607,E2 -27516.607} C_VEL
LIN {X 0,Y 141.005,Z 672.909,A -85,B 0,C 180,E1 -27518.673,E2 -27518.673} C_VEL
LIN {X 0,Y 138.739,Z 668.368,A -85,B 0,C 180,E1 -27521.925,E2 -27521.925} C_VEL
LIN {X 0,Y 136.142,Z 663.927,A -85,B 0,C 180,E1 -27526.567,E2 -27526.567} C_VEL
LIN {X 0,Y 134.173,Z 660.87,A -85,B 0,C 180,E1 -27531.718,E2 -27531.718} C_VEL
LIN {X 0,Y 133.054,Z 658.758,A -85,B 0,C 180,E1 -27538.487,E2 -27538.487} C_VEL
LIN {X 0,Y 132.998,Z 659.351,A -85,B 0,C 180,E1 -27541.93,E2 -27541.93} C_VEL
LIN {X 0,Y 133.634,Z 661.035,A -85,B 0,C 180,E1 -27546.796,E2 -27546.796} C_VEL
LIN {X 0,Y 134.987,Z 664.085,A -85,B 0,C 180,E1 -27551.449,E2 -27551.449} C_VEL
LIN {X 0,Y 137.093,Z 668.649,A -85,B 0,C 180,E1 -27556.09,E2 -27556.09} C_VEL
LIN {X 0,Y 138.844,Z 672.886,A -85,B 0,C 180,E1 -27559.113,E2 -27559.113} C_VEL
LIN {X 0,Y 141.097,Z 678.519,A -85,B 0,C 180,E1 -27562.366,E2 -27562.366} C_VEL
LIN {X 0,Y 143.36,Z 685.125,A -85,B 0,C 180,E1 -27565.256,E2 -27565.256} C_VEL
LIN {X 0,Y 143.96,Z 686.968,A -85,B 0,C 180,E1 -27565.967,E2 -27565.967} C_VEL
LIN {X 0,Y 138.291,Z 744.115,A -85,B 0,C 180,E1 -27567.932,E2 -27567.932} C_VEL
LIN {X 0,Y 135.719,Z 757.191,A -85,B 0,C 180,E1 -27568.704,E2 -27568.704} C_VEL
LIN {X 0,Y 132.215,Z 769.572,A -85,B 0,C 180,E1 -27569.873,E2 -27569.873} C_VEL
LIN {X 0,Y 128.364,Z 779.847,A -85,B 0,C 180,E1 -27571.184,E2 -27571.184} C_VEL
LIN {X 0,Y 123.587,Z 790.256,A -85,B 0,C 180,E1 -27572.984,E2 -27572.984} C_VEL
LIN {X 0,Y 117.532,Z 800.909,A -85,B 0,C 180,E1 -27575.436,E2 -27575.436} C_VEL
LIN {X 0,Y 110.549,Z 811.339,A -85,B 0,C 180,E1 -27578.847,E2 -27578.847} C_VEL
LIN {X 0,Y 103.466,Z 820.355,A -85,B 0,C 180,E1 -27583.095,E2 -27583.095} C_VEL
LIN {X 0,Y 96.958,Z 827.587,A -85,B 0,C 180,E1 -27587.892,E2 -27587.892} C_VEL
LIN {X 0,Y 90.088,Z 834.222,A -85,B 0,C 180,E1 -27594.187,E2 -27594.187} C_VEL
LIN {X 0,Y 85.287,Z 838.566,A -85,B 0,C 180,E1 -27600.364,E2 -27600.364} C_VEL
LIN {X 0,Y 82.626,Z 840.849,A -85,B 0,C 180,E1 -27604.827,E2 -27604.827} C_VEL
LIN {X 0,Y 80.463,Z 842.709,A -85,B 0,C 180,E1 -27609.547,E2 -27609.547} C_VEL
LIN {X 0,Y 78.811,Z 844.122,A -85,B 0,C 180,E1 -27614.479,E2 -27614.479} C_VEL
LIN {X 0,Y 77.692,Z 845.112,A -85,B 0,C 180,E1 -27619.572,E2 -27619.572} C_VEL
LIN {X 0,Y 77.054,Z 845.72,A -85,B 0,C 180,E1 -27624.763,E2 -27624.763} C_VEL
LIN {X 0,Y 76.884,Z 845.947,A -85,B 0,C 180,E1 -27629.996,E2 -27629.996} C_VEL
LIN {X 0,Y 77.69,Z 845.158,A -85,B 0,C 180,E1 -27640.419,E2 -27640.419} C_VEL
LIN {X 0,Y 78.806,Z 844.186,A -85,B 0,C 180,E1 -27645.513,E2 -27645.513} C_VEL
LIN {X 0,Y 80.453,Z 842.81,A -85,B 0,C 180,E1 -27650.447,E2 -27650.447} C_VEL
LIN {X 0,Y 83.845,Z 839.919,A -85,B 0,C 180,E1 -27657.448,E2 -27657.448} C_VEL
LIN {X 0,Y 88.268,Z 835.986,A -85,B 0,C 180,E1 -27663.867,E2 -27663.867} C_VEL
LIN {X 0,Y 93.804,Z 830.881,A -85,B 0,C 180,E1 -27669.551,E2 -27669.551} C_VEL
LIN {X 0,Y 100.034,Z 824.449,A -85,B 0,C 180,E1 -27674.627,E2 -27674.627} C_VEL
LIN {X 0,Y 106.854,Z 816.443,A -85,B 0,C 180,E1 -27679.137,E2 -27679.137} C_VEL
LIN {X 0,Y 113.172,Z 807.935,A -85,B 0,C 180,E1 -27682.591,E2 -27682.591} C_VEL
LIN {X 0,Y 114.241,Z 806.357,A -85,B 0,C 180,E1 -27683.1,E2 -27683.1} C_VEL
LIN {X 0,Y 112.152,Z 805.126,A -85,B 0,C 180,E1 -27685.668,E2 -27685.668} C_VEL
LIN {X 0,Y 108.296,Z 805.367,A -85,B 0,C 180,E1 -27688.723,E2 -27688.723} C_VEL
LIN {X 0,Y 100.73,Z 803.823,A -85,B 0,C 180,E1 -27699.582,E2 -27699.582} C_VEL
LIN {X 0,Y 97.949,Z 801.335,A -85,B 0,C 180,E1 -27711.749,E2 -27711.749} C_VEL
LIN {X 0,Y 98.99,Z 799.037,A -85,B 0,C 180,E1 -27720,E2 -27720} C_VEL
LIN {X 0,Y 104.612,Z 794.772,A -85,B 0,C 180,E1 -27731.627,E2 -27731.627} C_VEL
LIN {X 0,Y 111.761,Z 790.68,A -85,B 0,C 180,E1 -27739.405,E2 -27739.405} C_VEL
LIN {X 0,Y 115.816,Z 788.142,A -85,B 0,C 180,E1 -27742.288,E2 -27742.288} C_VEL
LIN {X 0,Y 126.199,Z 788.445,A -85,B 0,C 180,E1 -27746.456,E2 -27746.456} C_VEL
LIN {X 0,Y 133.441,Z 787.949,A -85,B 0,C 180,E1 -27748.811,E2 -27748.811} C_VEL
LIN {X 0,Y 131.768,Z 788.623,A -85,B 0,C 180,E1 -27749.74,E2 -27749.74} C_VEL
LIN {X 0,Y 124.539,Z 790.685,A -85,B 0,C 180,E1 -27751.794,E2 -27751.794} C_VEL
LIN {X 0,Y 118.649,Z 801.511,A -85,B 0,C 180,E1 -27753.983,E2 -27753.983} C_VEL
LIN {X 0,Y 112.047,Z 811.761,A -85,B 0,C 180,E1 -27756.902,E2 -27756.902} C_VEL
LIN {X 0,Y 104.579,Z 821.539,A -85,B 0,C 180,E1 -27760.891,E2 -27760.891} C_VEL
LIN {X 0,Y 97.766,Z 829.395,A -85,B 0,C 180,E1 -27765.509,E2 -27765.509} C_VEL
LIN {X 0,Y 92.714,Z 834.705,A -85,B 0,C 180,E1 -27769.89,E2 -27769.89} C_VEL
LIN {X 0,Y 87.228,Z 839.888,A -85,B 0,C 180,E1 -27775.673,E2 -27775.673} C_VEL
LIN {X 0,Y 82.779,Z 843.899,A -85,B 0,C 180,E1 -27782.168,E2 -27782.168} C_VEL
LIN {X 0,Y 79.558,Z 846.862,A -85,B 0,C 180,E1 -27789.312,E2 -27789.312} C_VEL
LIN {X 0,Y 78.071,Z 848.282,A -85,B 0,C 180,E1 -27794.337,E2 -27794.337} C_VEL
LIN {X 0,Y 76.81,Z 849.91,A -85,B 0,C 180,E1 -27804.755,E2 -27804.755} C_VEL
LIN {X 0,Y 76.915,Z 850.13,A -85,B 0,C 180,E1 -27810.004,E2 -27810.004} C_VEL
LIN {X 0,Y 76.811,Z 849.89,A -85,B 0,C 180,E1 -27815.254,E2 -27815.254} C_VEL
LIN {X 0,Y 78.071,Z 848.237,A -85,B 0,C 180,E1 -27825.672,E2 -27825.672} C_VEL
LIN {X 0,Y 79.551,Z 846.79,A -85,B 0,C 180,E1 -27830.698,E2 -27830.698} C_VEL
LIN {X 0,Y 82.759,Z 843.802,A -85,B 0,C 180,E1 -27837.848,E2 -27837.848} C_VEL
LIN {X 0,Y 87.19,Z 839.76,A -85,B 0,C 180,E1 -27844.354,E2 -27844.354} C_VEL
LIN {X 0,Y 92.697,Z 834.541,A -85,B 0,C 180,E1 -27850.128,E2 -27850.128} C_VEL
LIN {X 0,Y 96.014,Z 831.028,A -85,B 0,C 180,E1 -27853.145,E2 -27853.145} C_VEL
LIN {X 0,Y 98.467,Z 827.846,A -85,B 0,C 180,E1 -27855.694,E2 -27855.694} C_VEL
LIN {X 0,Y 101.334,Z 822.294,A -85,B 0,C 180,E1 -27860.119,E2 -27860.119} C_VEL
LIN {X 0,Y 104.5,Z 816.214,A -85,B 0,C 180,E1 -27864.088,E2 -27864.088} C_VEL
LIN {X 0,Y 107.265,Z 812.123,A -85,B 0,C 180,E1 -27865.858,E2 -27865.858} C_VEL
LIN {X 0,Y 114.121,Z 802.107,A -85,B 0,C 180,E1 -27868.706,E2 -27868.706} C_VEL
LIN {X 0,Y 120.571,Z 790.741,A -85,B 0,C 180,E1 -27870.971,E2 -27870.971} C_VEL
LIN {X 0,Y 125.692,Z 779.565,A -85,B 0,C 180,E1 -27872.582,E2 -27872.582} C_VEL
LIN {X 0,Y 130.18,Z 766.849,A -85,B 0,C 180,E1 -27873.84,E2 -27873.84} C_VEL
LIN {X 0,Y 133.472,Z 754.009,A -85,B 0,C 180,E1 -27874.663,E2 -27874.663} C_VEL
LIN {X 0,Y 135.443,Z 740.95,A -85,B 0,C 180,E1 -27875.249,E2 -27875.249} C_VEL
LIN {X 0,Y 139.147,Z 703.133,A -85,B 0,C 180,E1 -27876.543,E2 -27876.543} C_VEL
LIN {X 0,Y 139.911,Z 680.736,A -85,B 0,C 180,E1 -27878.739,E2 -27878.739} C_VEL
LIN {X 0,Y 137.051,Z 674.69,A -85,B 0,C 180,E1 -27883.069,E2 -27883.069} C_VEL
LIN {X 0,Y 134.845,Z 670.612,A -85,B 0,C 180,E1 -27887.394,E2 -27887.394} C_VEL
LIN {X 0,Y 133,Z 667.56,A -85,B 0,C 180,E1 -27892.79,E2 -27892.79} C_VEL
LIN {X 0,Y 132.188,Z 665.822,A -85,B 0,C 180,E1 -27898.477,E2 -27898.477} C_VEL
LIN {X 0,Y 132.161,Z 666.554,A -85,B 0,C 180,E1 -27902.495,E2 -27902.495} C_VEL
LIN {X 0,Y 132.877,Z 668.564,A -85,B 0,C 180,E1 -27907.407,E2 -27907.407} C_VEL
LIN {X 0,Y 134.223,Z 671.903,A -85,B 0,C 180,E1 -27911.898,E2 -27911.898} C_VEL
LIN {X 0,Y 135.783,Z 675.652,A -85,B 0,C 180,E1 -27915.467,E2 -27915.467} C_VEL
LIN {X 0,Y 137.121,Z 679.321,A -85,B 0,C 180,E1 -27918.007,E2 -27918.007} C_VEL
LIN {X 0,Y 139.088,Z 684.77,A -85,B 0,C 180,E1 -27921.147,E2 -27921.147} C_VEL
LIN {X 0,Y 140.696,Z 689.949,A -85,B 0,C 180,E1 -27923.452,E2 -27923.452} C_VEL
LIN {X 0,Y 135.219,Z 743.509,A -85,B 0,C 180,E1 -27925.249,E2 -27925.249} C_VEL
LIN {X 0,Y 132.65,Z 756.633,A -85,B 0,C 180,E1 -27925.965,E2 -27925.965} C_VEL
LIN {X 0,Y 128.831,Z 769.748,A -85,B 0,C 180,E1 -27927.138,E2 -27927.138} C_VEL
LIN {X 0,Y 124.843,Z 780.028,A -85,B 0,C 180,E1 -27928.401,E2 -27928.401} C_VEL
LIN {X 0,Y 119.881,Z 790.44,A -85,B 0,C 180,E1 -27930.146,E2 -27930.146} C_VEL
LIN {X 0,Y 113.565,Z 801.097,A -85,B 0,C 180,E1 -27932.518,E2 -27932.518} C_VEL
LIN {X 0,Y 106.232,Z 811.53,A -85,B 0,C 180,E1 -27935.858,E2 -27935.858} C_VEL
LIN {X 0,Y 99,Z 820.269,A -85,B 0,C 180,E1 -27939.926,E2 -27939.926} C_VEL
LIN {X 0,Y 91.824,Z 827.779,A -85,B 0,C 180,E1 -27944.925,E2 -27944.925} C_VEL
LIN {X 0,Y 84.432,Z 834.415,A -85,B 0,C 180,E1 -27951.366,E2 -27951.366} C_VEL
LIN {X 0,Y 79.174,Z 838.76,A -85,B 0,C 180,E1 -27957.814,E2 -27957.814} C_VEL
LIN {X 0,Y 76.24,Z 841.043,A -85,B 0,C 180,E1 -27962.55,E2 -27962.55} C_VEL
LIN {X 0,Y 73.845,Z 842.903,A -85,B 0,C 180,E1 -27967.619,E2 -27967.619} C_VEL
LIN {X 0,Y 72.006,Z 844.315,A -85,B 0,C 180,E1 -27972.969,E2 -27972.969} C_VEL
LIN {X 0,Y 69.999,Z 845.913,A -85,B 0,C 180,E1 -27984.233,E2 -27984.233} C_VEL
LIN {X 0,Y 69.785,Z 846.14,A -85,B 0,C 180,E1 -27989.995,E2 -27989.995} C_VEL
LIN {X 0,Y 69.94,Z 845.941,A -85,B 0,C 180,E1 -27995.762,E2 -27995.762} C_VEL
LIN {X 0,Y 70.708,Z 845.351,A -85,B 0,C 180,E1 -28001.461,E2 -28001.461} C_VEL
LIN {X 0,Y 72.001,Z 844.379,A -85,B 0,C 180,E1 -28007.022,E2 -28007.022} C_VEL
LIN {X 0,Y 73.835,Z 843.002,A -85,B 0,C 180,E1 -28012.374,E2 -28012.374} C_VEL
LIN {X 0,Y 77.604,Z 840.111,A -85,B 0,C 180,E1 -28019.868,E2 -28019.868} C_VEL
LIN {X 0,Y 82.46,Z 836.176,A -85,B 0,C 180,E1 -28026.621,E2 -28026.621} C_VEL
LIN {X 0,Y 88.443,Z 831.071,A -85,B 0,C 180,E1 -28032.482,E2 -28032.482} C_VEL
LIN {X 0,Y 95.107,Z 824.638,A -85,B 0,C 180,E1 -28037.636,E2 -28037.636} C_VEL
LIN {X 0,Y 102.342,Z 816.627,A -85,B 0,C 180,E1 -28042.153,E2 -28042.153} C_VEL
LIN {X 0,Y 106.686,Z 811.213,A -85,B 0,C 180,E1 -28044.44,E2 -28044.44} C_VEL
LIN {X 0,Y 106.694,Z 810.337,A -85,B 0,C 180,E1 -28045.285,E2 -28045.285} C_VEL
LIN {X 0,Y 104.14,Z 810.498,A -85,B 0,C 180,E1 -28047.324,E2 -28047.324} C_VEL
LIN {X 0,Y 94.667,Z 808.449,A -85,B 0,C 180,E1 -28062.725,E2 -28062.725} C_VEL
LIN {X 0,Y 93.504,Z 805.889,A -85,B 0,C 180,E1 -28075.689,E2 -28075.689} C_VEL
LIN {X 0,Y 97.897,Z 802.116,A -85,B 0,C 180,E1 -28088.255,E2 -28088.255} C_VEL
LIN {X 0,Y 103.387,Z 799.091,A -85,B 0,C 180,E1 -28095.778,E2 -28095.778} C_VEL
LIN {X 0,Y 110.762,Z 795.363,A -85,B 0,C 180,E1 -28102.377,E2 -28102.377} C_VEL
LIN {X 0,Y 115.046,Z 793.227,A -85,B 0,C 180,E1 -28105.317,E2 -28105.317} C_VEL
LIN {X 0,Y 119.642,Z 790.84,A -85,B 0,C 180,E1 -28108.03,E2 -28108.03} C_VEL
LIN {X 0,Y 120.579,Z 791.209,A -85,B 0,C 180,E1 -28109.047,E2 -28109.047} C_VEL
LIN {X 0,Y 114.126,Z 802.485,A -85,B 0,C 180,E1 -28111.31,E2 -28111.31} C_VEL
LIN {X 0,Y 107.93,Z 811.577,A -85,B 0,C 180,E1 -28113.885,E2 -28113.885} C_VEL
LIN {X 0,Y 100.056,Z 821.351,A -85,B 0,C 180,E1 -28117.802,E2 -28117.802} C_VEL
LIN {X 0,Y 92.813,Z 829.204,A -85,B 0,C 180,E1 -28122.42,E2 -28122.42} C_VEL
LIN {X 0,Y 87.368,Z 834.514,A -85,B 0,C 180,E1 -28126.869,E2 -28126.869} C_VEL
LIN {X 0,Y 81.43,Z 839.696,A -85,B 0,C 180,E1 -28132.838,E2 -28132.838} C_VEL
LIN {X 0,Y 76.552,Z 843.707,A -85,B 0,C 180,E1 -28139.678,E2 -28139.678} C_VEL
LIN {X 0,Y 72.923,Z 846.669,A -85,B 0,C 180,E1 -28147.331,E2 -28147.331} C_VEL
LIN {X 0,Y 71.235,Z 848.089,A -85,B 0,C 180,E1 -28152.789,E2 -28152.789} C_VEL
LIN {X 0,Y 69.743,Z 849.717,A -85,B 0,C 180,E1 -28164.221,E2 -28164.221} C_VEL
LIN {X 0,Y 69.82,Z 849.937,A -85,B 0,C 180,E1 -28170.005,E2 -28170.005} C_VEL
LIN {X 0,Y 69.744,Z 849.697,A -85,B 0,C 180,E1 -28175.788,E2 -28175.788} C_VEL
LIN {X 0,Y 71.235,Z 848.043,A -85,B 0,C 180,E1 -28187.221,E2 -28187.221} C_VEL
LIN {X 0,Y 72.917,Z 846.596,A -85,B 0,C 180,E1 -28192.682,E2 -28192.682} C_VEL
LIN {X 0,Y 76.532,Z 843.608,A -85,B 0,C 180,E1 -28200.34,E2 -28200.34} C_VEL
LIN {X 0,Y 81.398,Z 839.566,A -85,B 0,C 180,E1 -28207.189,E2 -28207.189} C_VEL
LIN {X 0,Y 88.154,Z 833.536,A -85,B 0,C 180,E1 -28213.93,E2 -28213.93} C_VEL
LIN {X 0,Y 95.092,Z 826.556,A -85,B 0,C 180,E1 -28219.253,E2 -28219.253} C_VEL
LIN {X 0,Y 102.581,Z 818.076,A -85,B 0,C 180,E1 -28223.616,E2 -28223.616} C_VEL
LIN {X 0,Y 107.265,Z 812.123,A -85,B 0,C 180,E1 -28225.858,E2 -28225.858} C_VEL
LIN {X 0,Y 108.972,Z 809.319,A -85,B 0,C 180,E1 -28227.067,E2 -28227.067} C_VEL
LIN {X 0,Y 110.523,Z 804.855,A -85,B 0,C 180,E1 -28229.606,E2 -28229.606} C_VEL
LIN {X 0,Y 112.072,Z 800.155,A -85,B 0,C 180,E1 -28231.975,E2 -28231.975} C_VEL
LIN {X 0,Y 113.664,Z 796.986,A -85,B 0,C 180,E1 -28232.892,E2 -28232.892} C_VEL
LIN {X 0,Y 119.527,Z 786.074,A -85,B 0,C 180,E1 -28234.697,E2 -28234.697} C_VEL
LIN {X 0,Y 124.494,Z 774.574,A -85,B 0,C 180,E1 -28236.044,E2 -28236.044} C_VEL
LIN {X 0,Y 128.577,Z 762.058,A -85,B 0,C 180,E1 -28237.03,E2 -28237.03} C_VEL
LIN {X 0,Y 131.516,Z 748.964,A -85,B 0,C 180,E1 -28237.701,E2 -28237.701} C_VEL
LIN {X 0,Y 133.841,Z 729.087,A -85,B 0,C 180,E1 -28238.414,E2 -28238.414} C_VEL
LIN {X 0,Y 136.407,Z 703.578,A -85,B 0,C 180,E1 -28239.278,E2 -28239.278} C_VEL
LIN {X 0,Y 137.227,Z 685.275,A -85,B 0,C 180,E1 -28241.09,E2 -28241.09} C_VEL
LIN {X 0,Y 135.352,Z 680.897,A -85,B 0,C 180,E1 -28244.364,E2 -28244.364} C_VEL
LIN {X 0,Y 133.571,Z 677.335,A -85,B 0,C 180,E1 -28248.236,E2 -28248.236} C_VEL
LIN {X 0,Y 132.06,Z 674.601,A -85,B 0,C 180,E1 -28253.027,E2 -28253.027} C_VEL
LIN {X 0,Y 131.321,Z 672.889,A -85,B 0,C 180,E1 -28258.467,E2 -28258.467} C_VEL
LIN {X 0,Y 131.363,Z 673.938,A -85,B 0,C 180,E1 -28263.451,E2 -28263.451} C_VEL
LIN {X 0,Y 132.071,Z 676.125,A -85,B 0,C 180,E1 -28267.837,E2 -28267.837} C_VEL
LIN {X 0,Y 133.708,Z 680.474,A -85,B 0,C 180,E1 -28272.997,E2 -28272.997} C_VEL
LIN {X 0,Y 135.09,Z 684.594,A -85,B 0,C 180,E1 -28276.141,E2 -28276.141} C_VEL
LIN {X 0,Y 136.85,Z 690.075,A -85,B 0,C 180,E1 -28279.403,E2 -28279.403} C_VEL
LIN {X 0,Y 137.713,Z 693.019,A -85,B 0,C 180,E1 -28280.833,E2 -28280.833} C_VEL
LIN {X 0,Y 132.299,Z 744.055,A -85,B 0,C 180,E1 -28282.493,E2 -28282.493} C_VEL
LIN {X 0,Y 129.702,Z 756.798,A -85,B 0,C 180,E1 -28283.148,E2 -28283.148} C_VEL
LIN {X 0,Y 125.758,Z 769.922,A -85,B 0,C 180,E1 -28284.264,E2 -28284.264} C_VEL
LIN {X 0,Y 120.893,Z 781.871,A -85,B 0,C 180,E1 -28285.695,E2 -28285.695} C_VEL
LIN {X 0,Y 114.99,Z 793.178,A -85,B 0,C 180,E1 -28287.594,E2 -28287.594} C_VEL
LIN {X 0,Y 108.488,Z 803.378,A -85,B 0,C 180,E1 -28289.947,E2 -28289.947} C_VEL
LIN {X 0,Y 102.234,Z 811.72,A -85,B 0,C 180,E1 -28292.631,E2 -28292.631} C_VEL
LIN {X 0,Y 95.595,Z 819.398,A -85,B 0,C 180,E1 -28296.026,E2 -28296.026} C_VEL
LIN {X 0,Y 88.14,Z 826.875,A -85,B 0,C 180,E1 -28300.751,E2 -28300.751} C_VEL
LIN {X 0,Y 81.173,Z 832.881,A -85,B 0,C 180,E1 -28306.155,E2 -28306.155} C_VEL
LIN {X 0,Y 75.041,Z 837.621,A -85,B 0,C 180,E1 -28312.495,E2 -28312.495} C_VEL
LIN {X 0,Y 70.001,Z 841.237,A -85,B 0,C 180,E1 -28319.863,E2 -28319.863} C_VEL
LIN {X 0,Y 67.334,Z 843.096,A -85,B 0,C 180,E1 -28325.318,E2 -28325.318} C_VEL
LIN {X 0,Y 65.243,Z 844.509,A -85,B 0,C 180,E1 -28331.141,E2 -28331.141} C_VEL
LIN {X 0,Y 62.94,Z 846.106,A -85,B 0,C 180,E1 -28343.584,E2 -28343.584} C_VEL
LIN {X 0,Y 62.7,Z 846.332,A -85,B 0,C 180,E1 -28349.995,E2 -28349.995} C_VEL
LIN {X 0,Y 62.897,Z 846.134,A -85,B 0,C 180,E1 -28356.41,E2 -28356.41} C_VEL
LIN {X 0,Y 63.76,Z 845.544,A -85,B 0,C 180,E1 -28362.73,E2 -28362.73} C_VEL
LIN {X 0,Y 65.238,Z 844.571,A -85,B 0,C 180,E1 -28368.85,E2 -28368.85} C_VEL
LIN {X 0,Y 67.323,Z 843.194,A -85,B 0,C 180,E1 -28374.675,E2 -28374.675} C_VEL
LIN {X 0,Y 71.529,Z 840.302,A -85,B 0,C 180,E1 -28382.704,E2 -28382.704} C_VEL
LIN {X 0,Y 76.876,Z 836.367,A -85,B 0,C 180,E1 -28389.781,E2 -28389.781} C_VEL
LIN {X 0,Y 83.345,Z 831.26,A -85,B 0,C 180,E1 -28395.781,E2 -28395.781} C_VEL
LIN {X 0,Y 90.476,Z 824.826,A -85,B 0,C 180,E1 -28400.96,E2 -28400.96} C_VEL
LIN {X 0,Y 98.005,Z 816.962,A -85,B 0,C 180,E1 -28405.363,E2 -28405.363} C_VEL
LIN {X 0,Y 98.959,Z 815.27,A -85,B 0,C 180,E1 -28406.619,E2 -28406.619} C_VEL
LIN {X 0,Y 89.834,Z 813.505,A -85,B 0,C 180,E1 -28421.764,E2 -28421.764} C_VEL
LIN {X 0,Y 88.561,Z 811.153,A -85,B 0,C 180,E1 -28435.448,E2 -28435.448} C_VEL
LIN {X 0,Y 93.162,Z 807.681,A -85,B 0,C 180,E1 -28448.678,E2 -28448.678} C_VEL
LIN {X 0,Y 102.588,Z 803.254,A -85,B 0,C 180,E1 -28460.031,E2 -28460.031} C_VEL
LIN {X 0,Y 112.414,Z 798.856,A -85,B 0,C 180,E1 -28467.052,E2 -28467.052} C_VEL
LIN {X 0,Y 112.079,Z 799.998,A -85,B 0,C 180,E1 -28467.669,E2 -28467.669} C_VEL
LIN {X 0,Y 105.554,Z 809.49,A -85,B 0,C 180,E1 -28470.061,E2 -28470.061} C_VEL
LIN {X 0,Y 98.557,Z 818.157,A -85,B 0,C 180,E1 -28473.09,E2 -28473.09} C_VEL
LIN {X 0,Y 90.643,Z 826.577,A -85,B 0,C 180,E1 -28477.377,E2 -28477.377} C_VEL
LIN {X 0,Y 82.81,Z 833.839,A -85,B 0,C 180,E1 -28482.985,E2 -28482.985} C_VEL
LIN {X 0,Y 75.868,Z 839.504,A -85,B 0,C 180,E1 -28489.582,E2 -28489.582} C_VEL
LIN {X 0,Y 70.499,Z 843.515,A -85,B 0,C 180,E1 -28496.756,E2 -28496.756} C_VEL
LIN {X 0,Y 66.381,Z 846.475,A -85,B 0,C 180,E1 -28504.951,E2 -28504.951} C_VEL
LIN {X 0,Y 64.469,Z 847.896,A -85,B 0,C 180,E1 -28510.917,E2 -28510.917} C_VEL
LIN {X 0,Y 62.656,Z 849.523,A -85,B 0,C 180,E1 -28523.565,E2 -28523.565} C_VEL
LIN {X 0,Y 62.717,Z 849.743,A -85,B 0,C 180,E1 -28530.005,E2 -28530.005} C_VEL
LIN {X 0,Y 62.657,Z 849.503,A -85,B 0,C 180,E1 -28536.446,E2 -28536.446} C_VEL
LIN {X 0,Y 64.469,Z 847.849,A -85,B 0,C 180,E1 -28549.094,E2 -28549.094} C_VEL
LIN {X 0,Y 66.374,Z 846.401,A -85,B 0,C 180,E1 -28555.063,E2 -28555.063} C_VEL
LIN {X 0,Y 70.48,Z 843.414,A -85,B 0,C 180,E1 -28563.265,E2 -28563.265} C_VEL
LIN {X 0,Y 75.843,Z 839.372,A -85,B 0,C 180,E1 -28570.445,E2 -28570.445} C_VEL
LIN {X 0,Y 82.542,Z 833.883,A -85,B 0,C 180,E1 -28576.842,E2 -28576.842} C_VEL
LIN {X 0,Y 90.592,Z 826.363,A -85,B 0,C 180,E1 -28582.677,E2 -28582.677} C_VEL
LIN {X 0,Y 98.526,Z 817.885,A -85,B 0,C 180,E1 -28586.949,E2 -28586.949} C_VEL
LIN {X 0,Y 105.531,Z 809.172,A -85,B 0,C 180,E1 -28589.974,E2 -28589.974} C_VEL
LIN {X 0,Y 112.805,Z 798.448,A -85,B 0,C 180,E1 -28592.603,E2 -28592.603} C_VEL
LIN {X 0,Y 113.664,Z 796.986,A -85,B 0,C 180,E1 -28592.892,E2 -28592.892} C_VEL
LIN {X 0,Y 116.127,Z 792.196,A -85,B 0,C 180,E1 -28594.023,E2 -28594.023} C_VEL
LIN {X 0,Y 118.979,Z 784.16,A -85,B 0,C 180,E1 -28596.474,E2 -28596.474} C_VEL
LIN {X 0,Y 121.502,Z 775.724,A -85,B 0,C 180,E1 -28598.679,E2 -28598.679} C_VEL
LIN {X 0,Y 123.313,Z 770.258,A -85,B 0,C 180,E1 -28599.435,E2 -28599.435} C_VEL
LIN {X 0,Y 127.166,Z 757.462,A -85,B 0,C 180,E1 -28600.244,E2 -28600.244} C_VEL
LIN {X 0,Y 129.584,Z 744.959,A -85,B 0,C 180,E1 -28600.784,E2 -28600.784} C_VEL
LIN {X 0,Y 133.968,Z 704.372,A -85,B 0,C 180,E1 -28602.083,E2 -28602.083} C_VEL
LIN {X 0,Y 134.755,Z 689.828,A -85,B 0,C 180,E1 -28603.567,E2 -28603.567} C_VEL
LIN {X 0,Y 133.703,Z 687.064,A -85,B 0,C 180,E1 -28605.736,E2 -28605.736} C_VEL
LIN {X 0,Y 132.261,Z 683.916,A -85,B 0,C 180,E1 -28609.282,E2 -28609.282} C_VEL
LIN {X 0,Y 130.929,Z 681.237,A -85,B 0,C 180,E1 -28614.224,E2 -28614.224} C_VEL
LIN {X 0,Y 130.453,Z 679.962,A -85,B 0,C 180,E1 -28618.457,E2 -28618.457} C_VEL
LIN {X 0,Y 130.457,Z 680.935,A -85,B 0,C 180,E1 -28623.088,E2 -28623.088} C_VEL
LIN {X 0,Y 131.096,Z 683.187,A -85,B 0,C 180,E1 -28627.509,E2 -28627.509} C_VEL
LIN {X 0,Y 132.505,Z 687.54,A -85,B 0,C 180,E1 -28632.394,E2 -28632.394} C_VEL
LIN {X 0,Y 133.631,Z 691.435,A -85,B 0,C 180,E1 -28635.246,E2 -28635.246} C_VEL
LIN {X 0,Y 135.024,Z 696.402,A -85,B 0,C 180,E1 -28638.149,E2 -28638.149} C_VEL
LIN {X 0,Y 129.687,Z 744.617,A -85,B 0,C 180,E1 -28639.611,E2 -28639.611} C_VEL
LIN {X 0,Y 126.889,Z 757.685,A -85,B 0,C 180,E1 -28640.257,E2 -28640.257} C_VEL
LIN {X 0,Y 123.019,Z 770.097,A -85,B 0,C 180,E1 -28641.258,E2 -28641.258} C_VEL
LIN {X 0,Y 118.749,Z 780.39,A -85,B 0,C 180,E1 -28642.365,E2 -28642.365} C_VEL
LIN {X 0,Y 113.427,Z 790.81,A -85,B 0,C 180,E1 -28643.942,E2 -28643.942} C_VEL
LIN {X 0,Y 106.626,Z 801.473,A -85,B 0,C 180,E1 -28646.09,E2 -28646.09} C_VEL
LIN {X 0,Y 98.582,Z 811.91,A -85,B 0,C 180,E1 -28649.149,E2 -28649.149} C_VEL
LIN {X 0,Y 91.145,Z 820.044,A -85,B 0,C 180,E1 -28652.667,E2 -28652.667} C_VEL
LIN {X 0,Y 83.673,Z 827.068,A -85,B 0,C 180,E1 -28657.061,E2 -28657.061} C_VEL
LIN {X 0,Y 76.206,Z 833.074,A -85,B 0,C 180,E1 -28662.451,E2 -28662.451} C_VEL
LIN {X 0,Y 69.531,Z 837.815,A -85,B 0,C 180,E1 -28668.923,E2 -28668.923} C_VEL
LIN {X 0,Y 63.953,Z 841.431,A -85,B 0,C 180,E1 -28676.664,E2 -28676.664} C_VEL
LIN {X 0,Y 60.96,Z 843.29,A -85,B 0,C 180,E1 -28682.533,E2 -28682.533} C_VEL
LIN {X 0,Y 58.572,Z 844.702,A -85,B 0,C 180,E1 -28688.896,E2 -28688.896} C_VEL
LIN {X 0,Y 55.908,Z 846.299,A -85,B 0,C 180,E1 -28702.773,E2 -28702.773} C_VEL
LIN {X 0,Y 55.609,Z 846.525,A -85,B 0,C 180,E1 -28709.994,E2 -28709.994} C_VEL
LIN {X 0,Y 55.848,Z 846.327,A -85,B 0,C 180,E1 -28717.223,E2 -28717.223} C_VEL
LIN {X 0,Y 56.863,Z 845.736,A -85,B 0,C 180,E1 -28724.305,E2 -28724.305} C_VEL
LIN {X 0,Y 58.567,Z 844.764,A -85,B 0,C 180,E1 -28731.094,E2 -28731.094} C_VEL
LIN {X 0,Y 60.949,Z 843.386,A -85,B 0,C 180,E1 -28737.46,E2 -28737.46} C_VEL
LIN {X 0,Y 65.663,Z 840.494,A -85,B 0,C 180,E1 -28746.056,E2 -28746.056} C_VEL
LIN {X 0,Y 71.565,Z 836.558,A -85,B 0,C 180,E1 -28753.42,E2 -28753.42} C_VEL
LIN {X 0,Y 78.56,Z 831.45,A -85,B 0,C 180,E1 -28759.493,E2 -28759.493} C_VEL
LIN {X 0,Y 86.183,Z 825.014,A -85,B 0,C 180,E1 -28764.626,E2 -28764.626} C_VEL
LIN {X 0,Y 91.533,Z 819.895,A -85,B 0,C 180,E1 -28767.62,E2 -28767.62} C_VEL
LIN {X 0,Y 89.009,Z 819.192,A -85,B 0,C 180,E1 -28771.722,E2 -28771.722} C_VEL
LIN {X 0,Y 83.609,Z 817.645,A -85,B 0,C 180,E1 -28785.394,E2 -28785.394} C_VEL
LIN {X 0,Y 84.329,Z 815.15,A -85,B 0,C 180,E1 -28800.121,E2 -28800.121} C_VEL
LIN {X 0,Y 90.923,Z 811.719,A -85,B 0,C 180,E1 -28813.408,E2 -28813.408} C_VEL
LIN {X 0,Y 102.288,Z 807.208,A -85,B 0,C 180,E1 -28824.346,E2 -28824.346} C_VEL
LIN {X 0,Y 103.453,Z 806.753,A -85,B 0,C 180,E1 -28825.158,E2 -28825.158} C_VEL
LIN {X 0,Y 103.146,Z 808.055,A -85,B 0,C 180,E1 -28826.264,E2 -28826.264} C_VEL
LIN {X 0,Y 94.858,Z 817.971,A -85,B 0,C 180,E1 -28829.486,E2 -28829.486} C_VEL
LIN {X 0,Y 86.494,Z 826.388,A -85,B 0,C 180,E1 -28833.615,E2 -28833.615} C_VEL
LIN {X 0,Y 78.671,Z 833.184,A -85,B 0,C 180,E1 -28838.707,E2 -28838.707} C_VEL
LIN {X 0,Y 72.855,Z 837.71,A -85,B 0,C 180,E1 -28843.664,E2 -28843.664} C_VEL
LIN {X 0,Y 66.531,Z 842.088,A -85,B 0,C 180,E1 -28850.676,E2 -28850.676} C_VEL
LIN {X 0,Y 62.909,Z 844.397,A -85,B 0,C 180,E1 -28856.049,E2 -28856.049} C_VEL
LIN {X 0,Y 59.981,Z 846.282,A -85,B 0,C 180,E1 -28862.058,E2 -28862.058} C_VEL
LIN {X 0,Y 57.778,Z 847.703,A -85,B 0,C 180,E1 -28868.604,E2 -28868.604} C_VEL
LIN {X 0,Y 55.589,Z 849.33,A -85,B 0,C 180,E1 -28882.743,E2 -28882.743} C_VEL
LIN {X 0,Y 55.612,Z 849.55,A -85,B 0,C 180,E1 -28890.006,E2 -28890.006} C_VEL
LIN {X 0,Y 55.59,Z 849.31,A -85,B 0,C 180,E1 -28897.269,E2 -28897.269} C_VEL
LIN {X 0,Y 57.778,Z 847.655,A -85,B 0,C 180,E1 -28911.408,E2 -28911.408} C_VEL
LIN {X 0,Y 59.973,Z 846.206,A -85,B 0,C 180,E1 -28917.958,E2 -28917.958} C_VEL
LIN {X 0,Y 64.649,Z 843.22,A -85,B 0,C 180,E1 -28926.726,E2 -28926.726} C_VEL
LIN {X 0,Y 70.576,Z 839.178,A -85,B 0,C 180,E1 -28934.198,E2 -28934.198} C_VEL
LIN {X 0,Y 78.57,Z 833.09,A -85,B 0,C 180,E1 -28941.234,E2 -28941.234} C_VEL
